LIN {X 0,Y 468.044,Z 554.979,A -85,B 0,C 180,E1 -7471.506,E2 -7471.506} C_VEL
LIN {X 0,Y 468.414,Z 546.131,A -85,B 0,C 180,E1 -7472.58,E2 -7472.58} C_VEL
LIN {X 0,Y 468.833,Z 536.407,A -85,B 0,C 180,E1 -7473.545,E2 -7473.545} C_VEL
LIN {X 0,Y 469.337,Z 525.651,A -85,B 0,C 180,E1 -7474.401,E2 -7474.401} C_VEL
LIN {X 0,Y 469.768,Z 513.644,A -85,B 0,C 180,E1 -7475.15,E2 -7475.15} C_VEL
LIN {X 0,Y 470.118,Z 501.093,A -85,B 0,C 180,E1 -7475.738,E2 -7475.738} C_VEL
LIN {X 0,Y 470.387,Z 488.653,A -85,B 0,C 180,E1 -7476.138,E2 -7476.138} C_VEL
LIN {X 0,Y 470.656,Z 471.073,A -85,B 0,C 180,E1 -7476.457,E2 -7476.457} C_VEL
LIN {X 0,Y 471.201,Z 391.14,A -85,B 0,C 180,E1 -7477.679,E2 -7477.679} C_VEL
LIN {X 0,Y 468.508,Z 378.211,A -85,B 0,C 180,E1 -7477.998,E2 -7477.998} C_VEL
LIN {X 0,Y 468.62,Z 369.536,A -85,B 0,C 180,E1 -7479.931,E2 -7479.931} C_VEL
LIN {X 0,Y 467.725,Z 363.226,A -85,B 0,C 180,E1 -7481.429,E2 -7481.429} C_VEL
LIN {X 0,Y 467.612,Z 363.236,A -85,B 0,C 180,E1 -7484.803,E2 -7484.803} C_VEL
LIN {X 0,Y 467.612,Z 363.233,A -85,B 0,C 180,E1 -7487.493,E2 -7487.493} C_VEL
LIN {X 0,Y 467.627,Z 363.237,A -85,B 0,C 180,E1 -7490.222,E2 -7490.222} C_VEL
LIN {X 0,Y 467.577,Z 363.241,A -85,B 0,C 180,E1 -7493.942,E2 -7493.942} C_VEL
LIN {X 0,Y 467.62,Z 363.234,A -85,B 0,C 180,E1 -7496.799,E2 -7496.799} C_VEL
LIN {X 0,Y 467.59,Z 363.239,A -85,B 0,C 180,E1 -7499.735,E2 -7499.735} C_VEL
LIN {X 0,Y 467.585,Z 363.239,A -85,B 0,C 180,E1 -7502.757,E2 -7502.757} C_VEL
LIN {X 0,Y 467.557,Z 363.244,A -85,B 0,C 180,E1 -7505.888,E2 -7505.888} C_VEL
LIN {X 0,Y 467.582,Z 363.239,A -85,B 0,C 180,E1 -7509.144,E2 -7509.144} C_VEL
LIN {X 0,Y 467.585,Z 363.239,A -85,B 0,C 180,E1 -7512.566,E2 -7512.566} C_VEL
LIN {X 0,Y 467.568,Z 363.241,A -85,B 0,C 180,E1 -7515.052,E2 -7515.052} C_VEL
LIN {X 0,Y 467.622,Z 363.235,A -85,B 0,C 180,E1 -7517.443,E2 -7517.443} C_VEL
LIN {X 0,Y 467.611,Z 363.236,A -85,B 0,C 180,E1 -7520.858,E2 -7520.858} C_VEL
LIN {X 0,Y 467.558,Z 363.244,A -85,B 0,C 180,E1 -7524.26,E2 -7524.26} C_VEL
LIN {X 0,Y 467.577,Z 363.241,A -85,B 0,C 180,E1 -7527.32,E2 -7527.32} C_VEL
LIN {X 0,Y 467.564,Z 363.242,A -85,B 0,C 180,E1 -7530.666,E2 -7530.666} C_VEL
LIN {X 0,Y 467.622,Z 363.236,A -85,B 0,C 180,E1 -7533.2,E2 -7533.2} C_VEL
LIN {X 0,Y 467.587,Z 363.239,A -85,B 0,C 180,E1 -7536.467,E2 -7536.467} C_VEL
LIN {X 0,Y 467.618,Z 363.238,A -85,B 0,C 180,E1 -7539.777,E2 -7539.777} C_VEL
LIN {X 0,Y 467.602,Z 363.238,A -85,B 0,C 180,E1 -7542.506,E2 -7542.506} C_VEL
LIN {X 0,Y 467.602,Z 363.239,A -85,B 0,C 180,E1 -7545.196,E2 -7545.196} C_VEL
LIN {X 0,Y 467.689,Z 363.228,A -85,B 0,C 180,E1 -7547.855,E2 -7547.855} C_VEL
LIN {X 0,Y 467.674,Z 363.23,A -85,B 0,C 180,E1 -7551.357,E2 -7551.357} C_VEL
LIN {X 0,Y 467.735,Z 363.221,A -85,B 0,C 180,E1 -7553.962,E2 -7553.962} C_VEL
LIN {X 0,Y 467.853,Z 363.208,A -85,B 0,C 180,E1 -7557.417,E2 -7557.417} C_VEL
LIN {X 0,Y 467.873,Z 363.203,A -85,B 0,C 180,E1 -7560,E2 -7560} C_VEL
LIN {X 0,Y 467.853,Z 363.209,A -85,B 0,C 180,E1 -7562.583,E2 -7562.583} C_VEL
LIN {X 0,Y 467.739,Z 363.22,A -85,B 0,C 180,E1 -7566.037,E2 -7566.037} C_VEL
LIN {X 0,Y 467.674,Z 363.231,A -85,B 0,C 180,E1 -7568.643,E2 -7568.643} C_VEL
LIN {X 0,Y 467.682,Z 363.23,A -85,B 0,C 180,E1 -7572.379,E2 -7572.379} C_VEL
LIN {X 0,Y 467.64,Z 363.232,A -85,B 0,C 180,E1 -7575.886,E2 -7575.886} C_VEL
LIN {X 0,Y 467.615,Z 363.236,A -85,B 0,C 180,E1 -7579.308,E2 -7579.308} C_VEL
LIN {X 0,Y 467.541,Z 363.246,A -85,B 0,C 180,E1 -7582.073,E2 -7582.073} C_VEL
LIN {X 0,Y 467.597,Z 363.238,A -85,B 0,C 180,E1 -7584.888,E2 -7584.888} C_VEL
LIN {X 0,Y 467.62,Z 363.235,A -85,B 0,C 180,E1 -7587.769,E2 -7587.769} C_VEL
LIN {X 0,Y 467.562,Z 363.242,A -85,B 0,C 180,E1 -7591.046,E2 -7591.046} C_VEL
LIN {X 0,Y 467.584,Z 363.244,A -85,B 0,C 180,E1 -7594.243,E2 -7594.243} C_VEL
LIN {X 0,Y 467.545,Z 363.243,A -85,B 0,C 180,E1 -7597.188,E2 -7597.188} C_VEL
LIN {X 0,Y 467.591,Z 363.242,A -85,B 0,C 180,E1 -7600.263,E2 -7600.263} C_VEL
LIN {X 0,Y 467.614,Z 363.236,A -85,B 0,C 180,E1 -7602.572,E2 -7602.572} C_VEL
LIN {X 0,Y 467.566,Z 363.24,A -85,B 0,C 180,E1 -7605.054,E2 -7605.054} C_VEL
LIN {X 0,Y 467.585,Z 363.238,A -85,B 0,C 180,E1 -7607.441,E2 -7607.441} C_VEL
LIN {X 0,Y 467.579,Z 363.238,A -85,B 0,C 180,E1 -7610.856,E2 -7610.856} C_VEL
LIN {X 0,Y 467.561,Z 363.243,A -85,B 0,C 180,E1 -7614.261,E2 -7614.261} C_VEL
LIN {X 0,Y 467.581,Z 363.238,A -85,B 0,C 180,E1 -7617.321,E2 -7617.321} C_VEL
LIN {X 0,Y 467.578,Z 363.24,A -85,B 0,C 180,E1 -7620.666,E2 -7620.666} C_VEL
LIN {X 0,Y 467.657,Z 363.297,A -85,B 0,C 180,E1 -7623.474,E2 -7623.474} C_VEL
LIN {X 0,Y 470.033,Z 375.942,A -85,B 0,C 180,E1 -7625.795,E2 -7625.795} C_VEL
LIN {X 0,Y 469.281,Z 393.239,A -85,B 0,C 180,E1 -7628.731,E2 -7628.731} C_VEL
LIN {X 0,Y 468.542,Z 411.912,A -85,B 0,C 180,E1 -7631.866,E2 -7631.866} C_VEL
LIN {X 0,Y 468.286,Z 419.154,A -85,B 0,C 180,E1 -7633.033,E2 -7633.033} C_VEL
LIN {X 0,Y 471.101,Z 439.527,A -85,B 0,C 180,E1 -7633.442,E2 -7633.442} C_VEL
LIN {X 0,Y 470.448,Z 528.104,A -85,B 0,C 180,E1 -7634.818,E2 -7634.818} C_VEL
LIN {X 0,Y 470.07,Z 541.203,A -85,B 0,C 180,E1 -7635.193,E2 -7635.193} C_VEL
LIN {X 0,Y 469.613,Z 553.288,A -85,B 0,C 180,E1 -7635.704,E2 -7635.704} C_VEL
LIN {X 0,Y 469.161,Z 564.699,A -85,B 0,C 180,E1 -7636.354,E2 -7636.354} C_VEL
LIN {X 0,Y 468.609,Z 576.212,A -85,B 0,C 180,E1 -7637.2,E2 -7637.2} C_VEL
LIN {X 0,Y 468.197,Z 587.011,A -85,B 0,C 180,E1 -7638.199,E2 -7638.199} C_VEL
LIN {X 0,Y 467.767,Z 595.641,A -85,B 0,C 180,E1 -7639.175,E2 -7639.175} C_VEL
LIN {X 0,Y 467.401,Z 603.6,A -85,B 0,C 180,E1 -7640.261,E2 -7640.261} C_VEL
LIN {X 0,Y 467.103,Z 611.375,A -85,B 0,C 180,E1 -7641.565,E2 -7641.565} C_VEL
LIN {X 0,Y 466.858,Z 618.527,A -85,B 0,C 180,E1 -7643.083,E2 -7643.083} C_VEL
LIN {X 0,Y 466.762,Z 623.289,A -85,B 0,C 180,E1 -7644.384,E2 -7644.384} C_VEL
LIN {X 0,Y 466.658,Z 626.925,A -85,B 0,C 180,E1 -7645.682,E2 -7645.682} C_VEL
LIN {X 0,Y 466.712,Z 628.806,A -85,B 0,C 180,E1 -7646.547,E2 -7646.547} C_VEL
LIN {X 0,Y 466.68,Z 630.213,A -85,B 0,C 180,E1 -7647.411,E2 -7647.411} C_VEL
LIN {X 0,Y 466.661,Z 631.215,A -85,B 0,C 180,E1 -7648.274,E2 -7648.274} C_VEL
LIN {X 0,Y 466.6,Z 632.044,A -85,B 0,C 180,E1 -7650,E2 -7650} C_VEL
LIN {X 0,Y 466.62,Z 631.83,A -85,B 0,C 180,E1 -7650.863,E2 -7650.863} C_VEL
LIN {X 0,Y 466.661,Z 631.221,A -85,B 0,C 180,E1 -7651.726,E2 -7651.726} C_VEL
LIN {X 0,Y 466.68,Z 630.222,A -85,B 0,C 180,E1 -7652.589,E2 -7652.589} C_VEL
LIN {X 0,Y 466.697,Z 628.821,A -85,B 0,C 180,E1 -7653.453,E2 -7653.453} C_VEL
LIN {X 0,Y 466.69,Z 625.873,A -85,B 0,C 180,E1 -7654.751,E2 -7654.751} C_VEL
LIN {X 0,Y 466.751,Z 621.888,A -85,B 0,C 180,E1 -7656.05,E2 -7656.05} C_VEL
LIN {X 0,Y 466.942,Z 615.771,A -85,B 0,C 180,E1 -7657.568,E2 -7657.568} C_VEL
LIN {X 0,Y 467.152,Z 609.091,A -85,B 0,C 180,E1 -7658.87,E2 -7658.87} C_VEL
LIN {X 0,Y 467.496,Z 600.812,A -85,B 0,C 180,E1 -7660.174,E2 -7660.174} C_VEL
LIN {X 0,Y 467.987,Z 592.352,A -85,B 0,C 180,E1 -7661.258,E2 -7661.258} C_VEL
LIN {X 0,Y 468.464,Z 582.434,A -85,B 0,C 180,E1 -7662.295,E2 -7662.295} C_VEL
LIN {X 0,Y 468.902,Z 571.605,A -85,B 0,C 180,E1 -7663.213,E2 -7663.213} C_VEL
LIN {X 0,Y 469.437,Z 560.342,A -85,B 0,C 180,E1 -7663.969,E2 -7663.969} C_VEL
LIN {X 0,Y 469.903,Z 548.916,A -85,B 0,C 180,E1 -7664.563,E2 -7664.563} C_VEL
LIN {X 0,Y 470.368,Z 535.882,A -85,B 0,C 180,E1 -7665.046,E2 -7665.046} C_VEL
LIN {X 0,Y 470.678,Z 521.948,A -85,B 0,C 180,E1 -7665.369,E2 -7665.369} C_VEL
LIN {X 0,Y 471.166,Z 437.424,A -85,B 0,C 180,E1 -7666.676,E2 -7666.676} C_VEL
LIN {X 0,Y 468.328,Z 418.62,A -85,B 0,C 180,E1 -7667.1,E2 -7667.1} C_VEL
LIN {X 0,Y 469.117,Z 400.586,A -85,B 0,C 180,E1 -7670.155,E2 -7670.155} C_VEL
LIN {X 0,Y 470.064,Z 380.743,A -85,B 0,C 180,E1 -7673.574,E2 -7673.574} C_VEL
LIN {X 0,Y 470.181,Z 375.849,A -85,B 0,C 180,E1 -7674.436,E2 -7674.436} C_VEL
LIN {X 0,Y 467.689,Z 363.253,A -85,B 0,C 180,E1 -7676.851,E2 -7676.851} C_VEL
LIN {X 0,Y 467.587,Z 363.239,A -85,B 0,C 180,E1 -7679.735,E2 -7679.735} C_VEL
LIN {X 0,Y 467.582,Z 363.239,A -85,B 0,C 180,E1 -7682.758,E2 -7682.758} C_VEL
LIN {X 0,Y 467.555,Z 363.247,A -85,B 0,C 180,E1 -7685.889,E2 -7685.889} C_VEL
LIN {X 0,Y 467.579,Z 363.238,A -85,B 0,C 180,E1 -7689.144,E2 -7689.144} C_VEL
LIN {X 0,Y 467.582,Z 363.236,A -85,B 0,C 180,E1 -7692.566,E2 -7692.566} C_VEL
LIN {X 0,Y 467.566,Z 363.238,A -85,B 0,C 180,E1 -7695.052,E2 -7695.052} C_VEL
LIN {X 0,Y 467.619,Z 363.235,A -85,B 0,C 180,E1 -7697.443,E2 -7697.443} C_VEL
LIN {X 0,Y 467.594,Z 363.234,A -85,B 0,C 180,E1 -7700.856,E2 -7700.856} C_VEL
LIN {X 0,Y 467.557,Z 363.24,A -85,B 0,C 180,E1 -7704.26,E2 -7704.26} C_VEL
LIN {X 0,Y 467.575,Z 363.243,A -85,B 0,C 180,E1 -7707.32,E2 -7707.32} C_VEL
LIN {X 0,Y 467.571,Z 363.238,A -85,B 0,C 180,E1 -7710.665,E2 -7710.665} C_VEL
LIN {X 0,Y 467.62,Z 363.236,A -85,B 0,C 180,E1 -7713.2,E2 -7713.2} C_VEL
LIN {X 0,Y 467.585,Z 363.231,A -85,B 0,C 180,E1 -7716.467,E2 -7716.467} C_VEL
LIN {X 0,Y 467.616,Z 363.233,A -85,B 0,C 180,E1 -7719.777,E2 -7719.777} C_VEL
LIN {X 0,Y 467.601,Z 363.235,A -85,B 0,C 180,E1 -7722.507,E2 -7722.507} C_VEL
LIN {X 0,Y 467.598,Z 363.238,A -85,B 0,C 180,E1 -7725.196,E2 -7725.196} C_VEL
LIN {X 0,Y 467.673,Z 363.226,A -85,B 0,C 180,E1 -7727.855,E2 -7727.855} C_VEL
LIN {X 0,Y 467.674,Z 363.23,A -85,B 0,C 180,E1 -7731.357,E2 -7731.357} C_VEL
LIN {X 0,Y 467.735,Z 363.214,A -85,B 0,C 180,E1 -7733.963,E2 -7733.963} C_VEL
LIN {X 0,Y 467.853,Z 363.204,A -85,B 0,C 180,E1 -7737.417,E2 -7737.417} C_VEL
LIN {X 0,Y 467.873,Z 363.2,A -85,B 0,C 180,E1 -7740,E2 -7740} C_VEL
LIN {X 0,Y 467.853,Z 363.208,A -85,B 0,C 180,E1 -7742.583,E2 -7742.583} C_VEL
LIN {X 0,Y 467.736,Z 363.219,A -85,B 0,C 180,E1 -7746.038,E2 -7746.038} C_VEL
LIN {X 0,Y 467.674,Z 363.228,A -85,B 0,C 180,E1 -7748.643,E2 -7748.643} C_VEL
LIN {X 0,Y 467.648,Z 363.23,A -85,B 0,C 180,E1 -7752.146,E2 -7752.146} C_VEL
LIN {X 0,Y 467.631,Z 363.231,A -85,B 0,C 180,E1 -7755.696,E2 -7755.696} C_VEL
LIN {X 0,Y 467.61,Z 363.238,A -85,B 0,C 180,E1 -7758.765,E2 -7758.765} C_VEL
LIN {X 0,Y 467.573,Z 363.236,A -85,B 0,C 180,E1 -7761.269,E2 -7761.269} C_VEL
LIN {X 0,Y 467.567,Z 363.242,A -85,B 0,C 180,E1 -7763.944,E2 -7763.944} C_VEL
LIN {X 0,Y 467.621,Z 363.228,A -85,B 0,C 180,E1 -7766.8,E2 -7766.8} C_VEL
LIN {X 0,Y 467.548,Z 363.243,A -85,B 0,C 180,E1 -7769.739,E2 -7769.739} C_VEL
LIN {X 0,Y 467.579,Z 363.239,A -85,B 0,C 180,E1 -7772.759,E2 -7772.759} C_VEL
LIN {X 0,Y 467.552,Z 363.246,A -85,B 0,C 180,E1 -7775.89,E2 -7775.89} C_VEL
LIN {X 0,Y 467.596,Z 363.236,A -85,B 0,C 180,E1 -7779.144,E2 -7779.144} C_VEL
LIN {X 0,Y 467.617,Z 363.234,A -85,B 0,C 180,E1 -7782.572,E2 -7782.572} C_VEL
LIN {X 0,Y 467.568,Z 363.243,A -85,B 0,C 180,E1 -7785.054,E2 -7785.054} C_VEL
LIN {X 0,Y 467.587,Z 363.241,A -85,B 0,C 180,E1 -7787.441,E2 -7787.441} C_VEL
LIN {X 0,Y 467.619,Z 363.235,A -85,B 0,C 180,E1 -7790.86,E2 -7790.86} C_VEL
LIN {X 0,Y 467.564,Z 363.244,A -85,B 0,C 180,E1 -7794.261,E2 -7794.261} C_VEL
LIN {X 0,Y 467.583,Z 363.241,A -85,B 0,C 180,E1 -7797.322,E2 -7797.322} C_VEL
LIN {X 0,Y 467.645,Z 363.312,A -85,B 0,C 180,E1 -7800.441,E2 -7800.441} C_VEL
LIN {X 0,Y 468.864,Z 370.492,A -85,B 0,C 180,E1 -7802.176,E2 -7802.176} C_VEL
LIN {X 0,Y 468.609,Z 378.685,A -85,B 0,C 180,E1 -7803.992,E2 -7803.992} C_VEL
LIN {X 0,Y 471.605,Z 392.631,A -85,B 0,C 180,E1 -7804.336,E2 -7804.336} C_VEL
LIN {X 0,Y 470.941,Z 465.261,A -85,B 0,C 180,E1 -7805.452,E2 -7805.452} C_VEL
LIN {X 0,Y 470.243,Z 471.119,A -85,B 0,C 180,E1 -7805.515,E2 -7805.515} C_VEL
LIN {X 0,Y 464.863,Z 488.149,A -85,B 0,C 180,E1 -7805.631,E2 -7805.631} C_VEL
LIN {X 0,Y 463.849,Z 493.862,A -85,B 0,C 180,E1 -7805.755,E2 -7805.755} C_VEL
LIN {X 0,Y 463.78,Z 495.764,A -85,B 0,C 180,E1 -7805.814,E2 -7805.814} C_VEL
LIN {X 0,Y 463.399,Z 507.867,A -85,B 0,C 180,E1 -7806.303,E2 -7806.303} C_VEL
LIN {X 0,Y 462.962,Z 520.228,A -85,B 0,C 180,E1 -7806.99,E2 -7806.99} C_VEL
LIN {X 0,Y 462.512,Z 531.401,A -85,B 0,C 180,E1 -7807.796,E2 -7807.796} C_VEL
LIN {X 0,Y 461.866,Z 542.532,A -85,B 0,C 180,E1 -7808.815,E2 -7808.815} C_VEL
LIN {X 0,Y 461.322,Z 552.494,A -85,B 0,C 180,E1 -7809.954,E2 -7809.954} C_VEL
LIN {X 0,Y 460.873,Z 560.782,A -85,B 0,C 180,E1 -7811.121,E2 -7811.121} C_VEL
LIN {X 0,Y 460.441,Z 568.432,A -85,B 0,C 180,E1 -7812.455,E2 -7812.455} C_VEL
LIN {X 0,Y 460.171,Z 573.745,A -85,B 0,C 180,E1 -7813.588,E2 -7813.588} C_VEL
LIN {X 0,Y 459.945,Z 578.843,A -85,B 0,C 180,E1 -7814.944,E2 -7814.944} C_VEL
LIN {X 0,Y 459.752,Z 582.757,A -85,B 0,C 180,E1 -7816.294,E2 -7816.294} C_VEL
LIN {X 0,Y 459.658,Z 586.366,A -85,B 0,C 180,E1 -7818.11,E2 -7818.11} C_VEL
LIN {X 0,Y 459.576,Z 587.863,A -85,B 0,C 180,E1 -7819.426,E2 -7819.426} C_VEL
LIN {X 0,Y 459.494,Z 588.394,A -85,B 0,C 180,E1 -7820.314,E2 -7820.314} C_VEL
LIN {X 0,Y 459.53,Z 588.483,A -85,B 0,C 180,E1 -7821.203,E2 -7821.203} C_VEL
LIN {X 0,Y 459.618,Z 587.497,A -85,B 0,C 180,E1 -7822.974,E2 -7822.974} C_VEL
LIN {X 0,Y 459.67,Z 586.415,A -85,B 0,C 180,E1 -7823.856,E2 -7823.856} C_VEL
LIN {X 0,Y 459.672,Z 584.89,A -85,B 0,C 180,E1 -7824.737,E2 -7824.737} C_VEL
LIN {X 0,Y 459.809,Z 581.826,A -85,B 0,C 180,E1 -7826.056,E2 -7826.056} C_VEL
LIN {X 0,Y 459.921,Z 577.728,A -85,B 0,C 180,E1 -7827.373,E2 -7827.373} C_VEL
LIN {X 0,Y 460.167,Z 571.478,A -85,B 0,C 180,E1 -7828.906,E2 -7828.906} C_VEL
LIN {X 0,Y 460.547,Z 564.676,A -85,B 0,C 180,E1 -7830.219,E2 -7830.219} C_VEL
LIN {X 0,Y 460.992,Z 556.186,A -85,B 0,C 180,E1 -7831.529,E2 -7831.529} C_VEL
LIN {X 0,Y 461.388,Z 547.502,A -85,B 0,C 180,E1 -7832.619,E2 -7832.619} C_VEL
LIN {X 0,Y 461.814,Z 537.987,A -85,B 0,C 180,E1 -7833.599,E2 -7833.599} C_VEL
LIN {X 0,Y 462.373,Z 527.564,A -85,B 0,C 180,E1 -7834.468,E2 -7834.468} C_VEL
LIN {X 0,Y 462.838,Z 516.054,A -85,B 0,C 180,E1 -7835.227,E2 -7835.227} C_VEL
LIN {X 0,Y 463.103,Z 504.183,A -85,B 0,C 180,E1 -7835.825,E2 -7835.825} C_VEL
LIN {X 0,Y 463.473,Z 491.224,A -85,B 0,C 180,E1 -7836.284,E2 -7836.284} C_VEL
LIN {X 0,Y 463.727,Z 478.883,A -85,B 0,C 180,E1 -7836.554,E2 -7836.554} C_VEL
LIN {X 0,Y 464.385,Z 392.218,A -85,B 0,C 180,E1 -7837.897,E2 -7837.897} C_VEL
LIN {X 0,Y 461.564,Z 378.518,A -85,B 0,C 180,E1 -7838.237,E2 -7838.237} C_VEL
LIN {X 0,Y 461.621,Z 370.343,A -85,B 0,C 180,E1 -7840.083,E2 -7840.083} C_VEL
LIN {X 0,Y 460.663,Z 364.106,A -85,B 0,C 180,E1 -7841.606,E2 -7841.606} C_VEL
LIN {X 0,Y 460.575,Z 364.111,A -85,B 0,C 180,E1 -7845.034,E2 -7845.034} C_VEL
LIN {X 0,Y 460.562,Z 364.113,A -85,B 0,C 180,E1 -7847.769,E2 -7847.769} C_VEL
LIN {X 0,Y 460.556,Z 364.117,A -85,B 0,C 180,E1 -7850.547,E2 -7850.547} C_VEL
LIN {X 0,Y 460.541,Z 364.116,A -85,B 0,C 180,E1 -7853.705,E2 -7853.705} C_VEL
LIN {X 0,Y 460.566,Z 364.118,A -85,B 0,C 180,E1 -7856.264,E2 -7856.264} C_VEL
LIN {X 0,Y 460.55,Z 364.114,A -85,B 0,C 180,E1 -7859.229,E2 -7859.229} C_VEL
LIN {X 0,Y 460.534,Z 364.122,A -85,B 0,C 180,E1 -7862.283,E2 -7862.283} C_VEL
LIN {X 0,Y 460.514,Z 364.119,A -85,B 0,C 180,E1 -7865.444,E2 -7865.444} C_VEL
LIN {X 0,Y 460.545,Z 364.115,A -85,B 0,C 180,E1 -7868.897,E2 -7868.897} C_VEL
LIN {X 0,Y 460.521,Z 364.123,A -85,B 0,C 180,E1 -7872.18,E2 -7872.18} C_VEL
LIN {X 0,Y 460.52,Z 364.119,A -85,B 0,C 180,E1 -7875.411,E2 -7875.411} C_VEL
LIN {X 0,Y 460.542,Z 364.117,A -85,B 0,C 180,E1 -7878.395,E2 -7878.395} C_VEL
LIN {X 0,Y 460.54,Z 364.117,A -85,B 0,C 180,E1 -7881.268,E2 -7881.268} C_VEL
LIN {X 0,Y 460.508,Z 364.121,A -85,B 0,C 180,E1 -7884.554,E2 -7884.554} C_VEL
LIN {X 0,Y 460.527,Z 364.121,A -85,B 0,C 180,E1 -7887.715,E2 -7887.715} C_VEL
LIN {X 0,Y 460.534,Z 364.118,A -85,B 0,C 180,E1 -7890.768,E2 -7890.768} C_VEL
LIN {X 0,Y 460.562,Z 364.117,A -85,B 0,C 180,E1 -7893.734,E2 -7893.734} C_VEL
LIN {X 0,Y 460.541,Z 364.117,A -85,B 0,C 180,E1 -7896.623,E2 -7896.623} C_VEL
LIN {X 0,Y 460.564,Z 364.115,A -85,B 0,C 180,E1 -7899.453,E2 -7899.453} C_VEL
LIN {X 0,Y 460.552,Z 364.116,A -85,B 0,C 180,E1 -7902.23,E2 -7902.23} C_VEL
LIN {X 0,Y 460.56,Z 364.116,A -85,B 0,C 180,E1 -7904.964,E2 -7904.964} C_VEL
LIN {X 0,Y 460.649,Z 364.106,A -85,B 0,C 180,E1 -7907.667,E2 -7907.667} C_VEL
LIN {X 0,Y 460.621,Z 364.108,A -85,B 0,C 180,E1 -7911.223,E2 -7911.223} C_VEL
LIN {X 0,Y 460.701,Z 364.098,A -85,B 0,C 180,E1 -7913.87,E2 -7913.87} C_VEL
LIN {X 0,Y 460.818,Z 364.084,A -85,B 0,C 180,E1 -7917.377,E2 -7917.377} C_VEL
LIN {X 0,Y 460.844,Z 364.079,A -85,B 0,C 180,E1 -7920,E2 -7920} C_VEL
LIN {X 0,Y 460.818,Z 364.085,A -85,B 0,C 180,E1 -7922.622,E2 -7922.622} C_VEL
LIN {X 0,Y 460.704,Z 364.097,A -85,B 0,C 180,E1 -7926.13,E2 -7926.13} C_VEL
LIN {X 0,Y 460.621,Z 364.109,A -85,B 0,C 180,E1 -7928.776,E2 -7928.776} C_VEL
LIN {X 0,Y 460.625,Z 364.11,A -85,B 0,C 180,E1 -7932.457,E2 -7932.457} C_VEL
LIN {X 0,Y 460.591,Z 364.111,A -85,B 0,C 180,E1 -7935.998,E2 -7935.998} C_VEL
LIN {X 0,Y 460.562,Z 364.115,A -85,B 0,C 180,E1 -7938.902,E2 -7938.902} C_VEL
LIN {X 0,Y 460.553,Z 364.115,A -85,B 0,C 180,E1 -7941.484,E2 -7941.484} C_VEL
LIN {X 0,Y 460.536,Z 364.121,A -85,B 0,C 180,E1 -7944.333,E2 -7944.333} C_VEL
LIN {X 0,Y 460.576,Z 364.113,A -85,B 0,C 180,E1 -7947.244,E2 -7947.244} C_VEL
LIN {X 0,Y 460.503,Z 364.126,A -85,B 0,C 180,E1 -7950.24,E2 -7950.24} C_VEL
LIN {X 0,Y 460.523,Z 364.118,A -85,B 0,C 180,E1 -7953.325,E2 -7953.325} C_VEL
LIN {X 0,Y 460.473,Z 364.126,A -85,B 0,C 180,E1 -7956.53,E2 -7956.53} C_VEL
LIN {X 0,Y 460.57,Z 364.115,A -85,B 0,C 180,E1 -7959.858,E2 -7959.858} C_VEL
LIN {X 0,Y 460.537,Z 364.116,A -85,B 0,C 180,E1 -7962.905,E2 -7962.905} C_VEL
LIN {X 0,Y 460.507,Z 364.123,A -85,B 0,C 180,E1 -7965.831,E2 -7965.831} C_VEL
LIN {X 0,Y 460.527,Z 364.117,A -85,B 0,C 180,E1 -7968.99,E2 -7968.99} C_VEL
LIN {X 0,Y 460.524,Z 364.117,A -85,B 0,C 180,E1 -7971.268,E2 -7971.268} C_VEL
LIN {X 0,Y 460.512,Z 364.119,A -85,B 0,C 180,E1 -7974.555,E2 -7974.555} C_VEL
LIN {X 0,Y 460.532,Z 364.12,A -85,B 0,C 180,E1 -7977.716,E2 -7977.716} C_VEL
LIN {X 0,Y 460.547,Z 364.116,A -85,B 0,C 180,E1 -7980.77,E2 -7980.77} C_VEL
LIN {X 0,Y 460.606,Z 364.146,A -85,B 0,C 180,E1 -7983.28,E2 -7983.28} C_VEL
LIN {X 0,Y 463.027,Z 376.596,A -85,B 0,C 180,E1 -7985.603,E2 -7985.603} C_VEL
LIN {X 0,Y 462.428,Z 392.07,A -85,B 0,C 180,E1 -7988.277,E2 -7988.277} C_VEL
LIN {X 0,Y 461.503,Z 412.791,A -85,B 0,C 180,E1 -7991.81,E2 -7991.81} C_VEL
LIN {X 0,Y 461.27,Z 418.674,A -85,B 0,C 180,E1 -7992.787,E2 -7992.787} C_VEL
LIN {X 0,Y 464.252,Z 439.85,A -85,B 0,C 180,E1 -7993.222,E2 -7993.222} C_VEL
LIN {X 0,Y 463.581,Z 526.961,A -85,B 0,C 180,E1 -7994.587,E2 -7994.587} C_VEL
LIN {X 0,Y 463.208,Z 540.34,A -85,B 0,C 180,E1 -7994.969,E2 -7994.969} C_VEL
LIN {X 0,Y 462.727,Z 552.571,A -85,B 0,C 180,E1 -7995.487,E2 -7995.487} C_VEL
LIN {X 0,Y 462.217,Z 564.087,A -85,B 0,C 180,E1 -7996.145,E2 -7996.145} C_VEL
LIN {X 0,Y 461.665,Z 575.364,A -85,B 0,C 180,E1 -7996.978,E2 -7996.978} C_VEL
LIN {X 0,Y 461.16,Z 586.507,A -85,B 0,C 180,E1 -7998.016,E2 -7998.016} C_VEL
LIN {X 0,Y 460.764,Z 595.173,A -85,B 0,C 180,E1 -7999.009,E2 -7999.009} C_VEL
LIN {X 0,Y 460.349,Z 603.157,A -85,B 0,C 180,E1 -8000.111,E2 -8000.111} C_VEL
LIN {X 0,Y 460.031,Z 610.965,A -85,B 0,C 180,E1 -8001.434,E2 -8001.434} C_VEL
LIN {X 0,Y 459.774,Z 618.134,A -85,B 0,C 180,E1 -8002.976,E2 -8002.976} C_VEL
LIN {X 0,Y 459.659,Z 622.91,A -85,B 0,C 180,E1 -8004.297,E2 -8004.297} C_VEL
LIN {X 0,Y 459.573,Z 626.56,A -85,B 0,C 180,E1 -8005.615,E2 -8005.615} C_VEL
LIN {X 0,Y 459.609,Z 628.448,A -85,B 0,C 180,E1 -8006.493,E2 -8006.493} C_VEL
LIN {X 0,Y 459.602,Z 629.864,A -85,B 0,C 180,E1 -8007.371,E2 -8007.371} C_VEL
LIN {X 0,Y 459.553,Z 631.486,A -85,B 0,C 180,E1 -8009.124,E2 -8009.124} C_VEL
LIN {X 0,Y 459.532,Z 631.711,A -85,B 0,C 180,E1 -8010,E2 -8010} C_VEL
LIN {X 0,Y 459.553,Z 631.504,A -85,B 0,C 180,E1 -8010.876,E2 -8010.876} C_VEL
LIN {X 0,Y 459.601,Z 629.904,A -85,B 0,C 180,E1 -8012.629,E2 -8012.629} C_VEL
LIN {X 0,Y 459.594,Z 628.508,A -85,B 0,C 180,E1 -8013.507,E2 -8013.507} C_VEL
LIN {X 0,Y 459.621,Z 625.57,A -85,B 0,C 180,E1 -8014.824,E2 -8014.824} C_VEL
LIN {X 0,Y 459.714,Z 620.574,A -85,B 0,C 180,E1 -8016.431,E2 -8016.431} C_VEL
LIN {X 0,Y 459.89,Z 614.487,A -85,B 0,C 180,E1 -8017.905,E2 -8017.905} C_VEL
LIN {X 0,Y 460.171,Z 607.602,A -85,B 0,C 180,E1 -8019.228,E2 -8019.228} C_VEL
LIN {X 0,Y 460.571,Z 599.022,A -85,B 0,C 180,E1 -8020.551,E2 -8020.551} C_VEL
LIN {X 0,Y 461.072,Z 590.225,A -85,B 0,C 180,E1 -8021.652,E2 -8021.652} C_VEL
LIN {X 0,Y 461.547,Z 579.698,A -85,B 0,C 180,E1 -8022.728,E2 -8022.728} C_VEL
LIN {X 0,Y 462.145,Z 568.617,A -85,B 0,C 180,E1 -8023.633,E2 -8023.633} C_VEL
LIN {X 0,Y 462.688,Z 556.514,A -85,B 0,C 180,E1 -8024.402,E2 -8024.402} C_VEL
LIN {X 0,Y 463.272,Z 543.889,A -85,B 0,C 180,E1 -8025.001,E2 -8025.001} C_VEL
LIN {X 0,Y 463.697,Z 531.564,A -85,B 0,C 180,E1 -8025.409,E2 -8025.409} C_VEL
LIN {X 0,Y 463.92,Z 515.932,A -85,B 0,C 180,E1 -8025.711,E2 -8025.711} C_VEL
LIN {X 0,Y 464.424,Z 438.295,A -85,B 0,C 180,E1 -8026.929,E2 -8026.929} C_VEL
LIN {X 0,Y 461.386,Z 418.289,A -85,B 0,C 180,E1 -8027.389,E2 -8027.389} C_VEL
LIN {X 0,Y 462.193,Z 400.426,A -85,B 0,C 180,E1 -8030.47,E2 -8030.47} C_VEL
LIN {X 0,Y 463.166,Z 381.944,A -85,B 0,C 180,E1 -8033.709,E2 -8033.709} C_VEL
LIN {X 0,Y 463.319,Z 377.648,A -85,B 0,C 180,E1 -8034.477,E2 -8034.477} C_VEL
LIN {X 0,Y 461.039,Z 366.113,A -85,B 0,C 180,E1 -8036.723,E2 -8036.723} C_VEL
LIN {X 0,Y 460.652,Z 364.106,A -85,B 0,C 180,E1 -8037.146,E2 -8037.146} C_VEL
LIN {X 0,Y 460.527,Z 364.12,A -85,B 0,C 180,E1 -8040.238,E2 -8040.238} C_VEL
LIN {X 0,Y 460.528,Z 364.118,A -85,B 0,C 180,E1 -8043.324,E2 -8043.324} C_VEL
LIN {X 0,Y 460.477,Z 364.125,A -85,B 0,C 180,E1 -8046.528,E2 -8046.528} C_VEL
LIN {X 0,Y 460.555,Z 364.118,A -85,B 0,C 180,E1 -8049.859,E2 -8049.859} C_VEL
LIN {X 0,Y 460.509,Z 364.117,A -85,B 0,C 180,E1 -8052.9,E2 -8052.9} C_VEL
LIN {X 0,Y 460.519,Z 364.121,A -85,B 0,C 180,E1 -8055.828,E2 -8055.828} C_VEL
LIN {X 0,Y 460.538,Z 364.113,A -85,B 0,C 180,E1 -8058.989,E2 -8058.989} C_VEL
LIN {X 0,Y 460.534,Z 364.116,A -85,B 0,C 180,E1 -8061.268,E2 -8061.268} C_VEL
LIN {X 0,Y 460.507,Z 364.117,A -85,B 0,C 180,E1 -8064.554,E2 -8064.554} C_VEL
LIN {X 0,Y 460.526,Z 364.122,A -85,B 0,C 180,E1 -8067.715,E2 -8067.715} C_VEL
LIN {X 0,Y 460.54,Z 364.114,A -85,B 0,C 180,E1 -8070.769,E2 -8070.769} C_VEL
LIN {X 0,Y 460.561,Z 364.106,A -85,B 0,C 180,E1 -8073.735,E2 -8073.735} C_VEL
LIN {X 0,Y 460.539,Z 364.109,A -85,B 0,C 180,E1 -8076.624,E2 -8076.624} C_VEL
LIN {X 0,Y 460.546,Z 364.117,A -85,B 0,C 180,E1 -8079.453,E2 -8079.453} C_VEL
LIN {X 0,Y 460.551,Z 364.113,A -85,B 0,C 180,E1 -8082.23,E2 -8082.23} C_VEL
LIN {X 0,Y 460.557,Z 364.115,A -85,B 0,C 180,E1 -8084.965,E2 -8084.965} C_VEL
LIN {X 0,Y 460.62,Z 364.105,A -85,B 0,C 180,E1 -8087.666,E2 -8087.666} C_VEL
LIN {X 0,Y 460.621,Z 364.11,A -85,B 0,C 180,E1 -8091.224,E2 -8091.224} C_VEL
LIN {X 0,Y 460.701,Z 364.09,A -85,B 0,C 180,E1 -8093.87,E2 -8093.87} C_VEL
LIN {X 0,Y 460.818,Z 364.08,A -85,B 0,C 180,E1 -8097.378,E2 -8097.378} C_VEL
LIN {X 0,Y 460.844,Z 364.075,A -85,B 0,C 180,E1 -8100,E2 -8100} C_VEL
LIN {X 0,Y 460.818,Z 364.085,A -85,B 0,C 180,E1 -8102.623,E2 -8102.623} C_VEL
LIN {X 0,Y 460.702,Z 364.096,A -85,B 0,C 180,E1 -8106.13,E2 -8106.13} C_VEL
LIN {X 0,Y 460.621,Z 364.108,A -85,B 0,C 180,E1 -8108.777,E2 -8108.777} C_VEL
LIN {X 0,Y 460.605,Z 364.109,A -85,B 0,C 180,E1 -8112.445,E2 -8112.445} C_VEL
LIN {X 0,Y 460.592,Z 364.109,A -85,B 0,C 180,E1 -8115.998,E2 -8115.998} C_VEL
LIN {X 0,Y 460.563,Z 364.114,A -85,B 0,C 180,E1 -8118.903,E2 -8118.903} C_VEL
LIN {X 0,Y 460.509,Z 364.116,A -85,B 0,C 180,E1 -8121.486,E2 -8121.486} C_VEL
LIN {X 0,Y 460.536,Z 364.118,A -85,B 0,C 180,E1 -8124.333,E2 -8124.333} C_VEL
LIN {X 0,Y 460.577,Z 364.103,A -85,B 0,C 180,E1 -8127.244,E2 -8127.244} C_VEL
LIN {X 0,Y 460.505,Z 364.125,A -85,B 0,C 180,E1 -8130.241,E2 -8130.241} C_VEL
LIN {X 0,Y 460.525,Z 364.117,A -85,B 0,C 180,E1 -8133.326,E2 -8133.326} C_VEL
LIN {X 0,Y 460.475,Z 364.126,A -85,B 0,C 180,E1 -8136.53,E2 -8136.53} C_VEL
LIN {X 0,Y 460.571,Z 364.116,A -85,B 0,C 180,E1 -8139.859,E2 -8139.859} C_VEL
LIN {X 0,Y 460.54,Z 364.115,A -85,B 0,C 180,E1 -8142.905,E2 -8142.905} C_VEL
LIN {X 0,Y 460.509,Z 364.124,A -85,B 0,C 180,E1 -8145.831,E2 -8145.831} C_VEL
LIN {X 0,Y 460.538,Z 364.118,A -85,B 0,C 180,E1 -8148.991,E2 -8148.991} C_VEL
LIN {X 0,Y 460.547,Z 364.118,A -85,B 0,C 180,E1 -8151.27,E2 -8151.27} C_VEL
LIN {X 0,Y 460.515,Z 364.12,A -85,B 0,C 180,E1 -8154.556,E2 -8154.556} C_VEL
LIN {X 0,Y 460.533,Z 364.122,A -85,B 0,C 180,E1 -8157.717,E2 -8157.717} C_VEL
LIN {X 0,Y 460.607,Z 364.241,A -85,B 0,C 180,E1 -8160.231,E2 -8160.231} C_VEL
LIN {X 0,Y 461.84,Z 371.277,A -85,B 0,C 180,E1 -8161.96,E2 -8161.96} C_VEL
LIN {X 0,Y 461.681,Z 378.848,A -85,B 0,C 180,E1 -8163.699,E2 -8163.699} C_VEL
LIN {X 0,Y 464.892,Z 393.973,A -85,B 0,C 180,E1 -8164.08,E2 -8164.08} C_VEL
LIN {X 0,Y 463.956,Z 485.671,A -85,B 0,C 180,E1 -8165.534,E2 -8165.534} C_VEL
LIN {X 0,Y 463.78,Z 495.764,A -85,B 0,C 180,E1 -8165.814,E2 -8165.814} C_VEL
LIN {X 0,Y 463.118,Z 501.433,A -85,B 0,C 180,E1 -8165.999,E2 -8165.999} C_VEL
LIN {X 0,Y 460.095,Z 510.546,A -85,B 0,C 180,E1 -8166.304,E2 -8166.304} C_VEL
LIN {X 0,Y 456.903,Z 519.371,A -85,B 0,C 180,E1 -8166.7,E2 -8166.7} C_VEL
LIN {X 0,Y 455.983,Z 524.587,A -85,B 0,C 180,E1 -8167.024,E2 -8167.024} C_VEL
LIN {X 0,Y 455.38,Z 535.978,A -85,B 0,C 180,E1 -8167.934,E2 -8167.934} C_VEL
LIN {X 0,Y 454.781,Z 546.065,A -85,B 0,C 180,E1 -8168.944,E2 -8168.944} C_VEL
LIN {X 0,Y 454.232,Z 555.372,A -85,B 0,C 180,E1 -8170.1,E2 -8170.1} C_VEL
LIN {X 0,Y 453.718,Z 564.383,A -85,B 0,C 180,E1 -8171.486,E2 -8171.486} C_VEL
LIN {X 0,Y 453.301,Z 571.518,A -85,B 0,C 180,E1 -8172.868,E2 -8172.868} C_VEL
LIN {X 0,Y 452.956,Z 577.765,A -85,B 0,C 180,E1 -8174.414,E2 -8174.414} C_VEL
LIN {X 0,Y 452.712,Z 582.803,A -85,B 0,C 180,E1 -8176.077,E2 -8176.077} C_VEL
LIN {X 0,Y 452.62,Z 585.737,A -85,B 0,C 180,E1 -8177.445,E2 -8177.445} C_VEL
LIN {X 0,Y 452.573,Z 587.115,A -85,B 0,C 180,E1 -8178.354,E2 -8178.354} C_VEL
LIN {X 0,Y 452.506,Z 588.089,A -85,B 0,C 180,E1 -8179.259,E2 -8179.259} C_VEL
LIN {X 0,Y 452.412,Z 588.673,A -85,B 0,C 180,E1 -8180.161,E2 -8180.161} C_VEL
LIN {X 0,Y 452.439,Z 588.839,A -85,B 0,C 180,E1 -8181.064,E2 -8181.064} C_VEL
LIN {X 0,Y 452.535,Z 587.938,A -85,B 0,C 180,E1 -8182.863,E2 -8182.863} C_VEL
LIN {X 0,Y 452.587,Z 586.911,A -85,B 0,C 180,E1 -8183.76,E2 -8183.76} C_VEL
LIN {X 0,Y 452.603,Z 585.461,A -85,B 0,C 180,E1 -8184.654,E2 -8184.654} C_VEL
LIN {X 0,Y 452.726,Z 582.489,A -85,B 0,C 180,E1 -8185.994,E2 -8185.994} C_VEL
LIN {X 0,Y 452.859,Z 578.486,A -85,B 0,C 180,E1 -8187.332,E2 -8187.332} C_VEL
LIN {X 0,Y 453.021,Z 573.343,A -85,B 0,C 180,E1 -8188.667,E2 -8188.667} C_VEL
LIN {X 0,Y 453.454,Z 566.868,A -85,B 0,C 180,E1 -8190,E2 -8190} C_VEL
LIN {X 0,Y 453.862,Z 558.854,A -85,B 0,C 180,E1 -8191.331,E2 -8191.331} C_VEL
LIN {X 0,Y 454.271,Z 550.681,A -85,B 0,C 180,E1 -8192.438,E2 -8192.438} C_VEL
LIN {X 0,Y 454.728,Z 540.697,A -85,B 0,C 180,E1 -8193.544,E2 -8193.544} C_VEL
LIN {X 0,Y 455.351,Z 529.374,A -85,B 0,C 180,E1 -8194.537,E2 -8194.537} C_VEL
LIN {X 0,Y 455.886,Z 518.274,A -85,B 0,C 180,E1 -8195.307,E2 -8195.307} C_VEL
LIN {X 0,Y 456.195,Z 507.092,A -85,B 0,C 180,E1 -8195.913,E2 -8195.913} C_VEL
LIN {X 0,Y 456.519,Z 494.417,A -85,B 0,C 180,E1 -8196.408,E2 -8196.408} C_VEL
LIN {X 0,Y 456.821,Z 480.979,A -85,B 0,C 180,E1 -8196.737,E2 -8196.737} C_VEL
LIN {X 0,Y 457.581,Z 393.227,A -85,B 0,C 180,E1 -8198.118,E2 -8198.118} C_VEL
LIN {X 0,Y 454.615,Z 378.81,A -85,B 0,C 180,E1 -8198.484,E2 -8198.484} C_VEL
LIN {X 0,Y 454.589,Z 371.139,A -85,B 0,C 180,E1 -8200.241,E2 -8200.241} C_VEL
LIN {X 0,Y 453.61,Z 364.985,A -85,B 0,C 180,E1 -8201.725,E2 -8201.725} C_VEL
LIN {X 0,Y 453.555,Z 364.984,A -85,B 0,C 180,E1 -8205.273,E2 -8205.273} C_VEL
LIN {X 0,Y 453.515,Z 364.992,A -85,B 0,C 180,E1 -8208.055,E2 -8208.055} C_VEL
LIN {X 0,Y 453.487,Z 364.995,A -85,B 0,C 180,E1 -8210.882,E2 -8210.882} C_VEL
LIN {X 0,Y 453.504,Z 364.993,A -85,B 0,C 180,E1 -8213.888,E2 -8213.888} C_VEL
LIN {X 0,Y 453.512,Z 364.992,A -85,B 0,C 180,E1 -8216.705,E2 -8216.705} C_VEL
LIN {X 0,Y 453.491,Z 364.995,A -85,B 0,C 180,E1 -8219.788,E2 -8219.788} C_VEL
LIN {X 0,Y 453.492,Z 364.994,A -85,B 0,C 180,E1 -8223.188,E2 -8223.188} C_VEL
LIN {X 0,Y 453.456,Z 365.002,A -85,B 0,C 180,E1 -8226.299,E2 -8226.299} C_VEL
LIN {X 0,Y 453.489,Z 364.995,A -85,B 0,C 180,E1 -8229.449,E2 -8229.449} C_VEL
LIN {X 0,Y 453.475,Z 365,A -85,B 0,C 180,E1 -8231.934,E2 -8231.934} C_VEL
LIN {X 0,Y 453.491,Z 364.995,A -85,B 0,C 180,E1 -8235.469,E2 -8235.469} C_VEL
LIN {X 0,Y 453.494,Z 364.997,A -85,B 0,C 180,E1 -8238.21,E2 -8238.21} C_VEL
LIN {X 0,Y 453.527,Z 364.99,A -85,B 0,C 180,E1 -8240.787,E2 -8240.787} C_VEL
LIN {X 0,Y 453.452,Z 365.003,A -85,B 0,C 180,E1 -8243.916,E2 -8243.916} C_VEL
LIN {X 0,Y 453.478,Z 364.997,A -85,B 0,C 180,E1 -8247.15,E2 -8247.15} C_VEL
LIN {X 0,Y 453.469,Z 364.999,A -85,B 0,C 180,E1 -8250.267,E2 -8250.267} C_VEL
LIN {X 0,Y 453.508,Z 364.994,A -85,B 0,C 180,E1 -8253.294,E2 -8253.294} C_VEL
LIN {X 0,Y 453.498,Z 364.995,A -85,B 0,C 180,E1 -8256.238,E2 -8256.238} C_VEL
LIN {X 0,Y 453.5,Z 364.995,A -85,B 0,C 180,E1 -8259.118,E2 -8259.118} C_VEL
LIN {X 0,Y 453.504,Z 364.995,A -85,B 0,C 180,E1 -8261.944,E2 -8261.944} C_VEL
LIN {X 0,Y 453.533,Z 364.992,A -85,B 0,C 180,E1 -8264.726,E2 -8264.726} C_VEL
LIN {X 0,Y 453.594,Z 364.984,A -85,B 0,C 180,E1 -8267.472,E2 -8267.472} C_VEL
LIN {X 0,Y 453.585,Z 364.984,A -85,B 0,C 180,E1 -8271.086,E2 -8271.086} C_VEL
LIN {X 0,Y 453.669,Z 364.974,A -85,B 0,C 180,E1 -8273.774,E2 -8273.774} C_VEL
LIN {X 0,Y 453.758,Z 364.963,A -85,B 0,C 180,E1 -8277.337,E2 -8277.337} C_VEL
LIN {X 0,Y 453.815,Z 364.955,A -85,B 0,C 180,E1 -8280,E2 -8280} C_VEL
LIN {X 0,Y 453.758,Z 364.964,A -85,B 0,C 180,E1 -8282.663,E2 -8282.663} C_VEL
LIN {X 0,Y 453.671,Z 364.974,A -85,B 0,C 180,E1 -8286.225,E2 -8286.225} C_VEL
LIN {X 0,Y 453.585,Z 364.984,A -85,B 0,C 180,E1 -8288.913,E2 -8288.913} C_VEL
LIN {X 0,Y 453.593,Z 364.985,A -85,B 0,C 180,E1 -8292.551,E2 -8292.551} C_VEL
LIN {X 0,Y 453.536,Z 364.992,A -85,B 0,C 180,E1 -8296.196,E2 -8296.196} C_VEL
LIN {X 0,Y 453.512,Z 364.993,A -85,B 0,C 180,E1 -8299.041,E2 -8299.041} C_VEL
LIN {X 0,Y 453.49,Z 364.996,A -85,B 0,C 180,E1 -8301.835,E2 -8301.835} C_VEL
LIN {X 0,Y 453.507,Z 364.994,A -85,B 0,C 180,E1 -8304.735,E2 -8304.735} C_VEL
LIN {X 0,Y 453.53,Z 364.992,A -85,B 0,C 180,E1 -8307.961,E2 -8307.961} C_VEL
LIN {X 0,Y 453.459,Z 364.999,A -85,B 0,C 180,E1 -8311.526,E2 -8311.526} C_VEL
LIN {X 0,Y 453.483,Z 364.996,A -85,B 0,C 180,E1 -8314.778,E2 -8314.778} C_VEL
LIN {X 0,Y 453.478,Z 364.999,A -85,B 0,C 180,E1 -8318.31,E2 -8318.31} C_VEL
LIN {X 0,Y 453.511,Z 364.992,A -85,B 0,C 180,E1 -8320.607,E2 -8320.607} C_VEL
LIN {X 0,Y 453.477,Z 364.996,A -85,B 0,C 180,E1 -8323.248,E2 -8323.248} C_VEL
LIN {X 0,Y 453.462,Z 365,A -85,B 0,C 180,E1 -8325.78,E2 -8325.78} C_VEL
LIN {X 0,Y 453.475,Z 364.999,A -85,B 0,C 180,E1 -8328.21,E2 -8328.21} C_VEL
LIN {X 0,Y 453.491,Z 364.993,A -85,B 0,C 180,E1 -8330.794,E2 -8330.794} C_VEL
LIN {X 0,Y 453.455,Z 365.004,A -85,B 0,C 180,E1 -8333.918,E2 -8333.918} C_VEL
LIN {X 0,Y 453.482,Z 364.994,A -85,B 0,C 180,E1 -8337.152,E2 -8337.152} C_VEL
LIN {X 0,Y 453.513,Z 364.997,A -85,B 0,C 180,E1 -8340.272,E2 -8340.272} C_VEL
LIN {X 0,Y 453.59,Z 365.175,A -85,B 0,C 180,E1 -8343.113,E2 -8343.113} C_VEL
LIN {X 0,Y 456.078,Z 378.052,A -85,B 0,C 180,E1 -8345.554,E2 -8345.554} C_VEL
LIN {X 0,Y 455.418,Z 393.5,A -85,B 0,C 180,E1 -8348.262,E2 -8348.262} C_VEL
LIN {X 0,Y 454.482,Z 413.659,A -85,B 0,C 180,E1 -8351.752,E2 -8351.752} C_VEL
LIN {X 0,Y 454.303,Z 418.353,A -85,B 0,C 180,E1 -8352.542,E2 -8352.542} C_VEL
LIN {X 0,Y 457.402,Z 439.991,A -85,B 0,C 180,E1 -8352.996,E2 -8352.996} C_VEL
LIN {X 0,Y 456.698,Z 526.846,A -85,B 0,C 180,E1 -8354.378,E2 -8354.378} C_VEL
LIN {X 0,Y 456.313,Z 540.155,A -85,B 0,C 180,E1 -8354.765,E2 -8354.765} C_VEL
LIN {X 0,Y 455.769,Z 552.92,A -85,B 0,C 180,E1 -8355.318,E2 -8355.318} C_VEL
LIN {X 0,Y 455.207,Z 565.055,A -85,B 0,C 180,E1 -8356.041,E2 -8356.041} C_VEL
LIN {X 0,Y 454.572,Z 577.315,A -85,B 0,C 180,E1 -8356.993,E2 -8356.993} C_VEL
LIN {X 0,Y 454.107,Z 588.071,A -85,B 0,C 180,E1 -8358.054,E2 -8358.054} C_VEL
LIN {X 0,Y 453.54,Z 598.053,A -85,B 0,C 180,E1 -8359.284,E2 -8359.284} C_VEL
LIN {X 0,Y 453.109,Z 606.84,A -85,B 0,C 180,E1 -8360.627,E2 -8360.627} C_VEL
LIN {X 0,Y 452.837,Z 613.846,A -85,B 0,C 180,E1 -8361.971,E2 -8361.971} C_VEL
LIN {X 0,Y 452.634,Z 619.457,A -85,B 0,C 180,E1 -8363.313,E2 -8363.313} C_VEL
LIN {X 0,Y 452.578,Z 623.861,A -85,B 0,C 180,E1 -8364.654,E2 -8364.654} C_VEL
LIN {X 0,Y 452.494,Z 626.186,A -85,B 0,C 180,E1 -8365.546,E2 -8365.546} C_VEL
LIN {X 0,Y 452.507,Z 628.081,A -85,B 0,C 180,E1 -8366.438,E2 -8366.438} C_VEL
LIN {X 0,Y 452.525,Z 629.51,A -85,B 0,C 180,E1 -8367.33,E2 -8367.33} C_VEL
LIN {X 0,Y 452.488,Z 631.145,A -85,B 0,C 180,E1 -8369.11,E2 -8369.11} C_VEL
LIN {X 0,Y 452.465,Z 631.377,A -85,B 0,C 180,E1 -8370,E2 -8370} C_VEL
LIN {X 0,Y 452.488,Z 631.18,A -85,B 0,C 180,E1 -8370.89,E2 -8370.89} C_VEL
LIN {X 0,Y 452.523,Z 629.591,A -85,B 0,C 180,E1 -8372.67,E2 -8372.67} C_VEL
LIN {X 0,Y 452.492,Z 628.202,A -85,B 0,C 180,E1 -8373.562,E2 -8373.562} C_VEL
LIN {X 0,Y 452.551,Z 625.277,A -85,B 0,C 180,E1 -8374.9,E2 -8374.9} C_VEL
LIN {X 0,Y 452.61,Z 620.797,A -85,B 0,C 180,E1 -8376.396,E2 -8376.396} C_VEL
LIN {X 0,Y 452.778,Z 616.232,A -85,B 0,C 180,E1 -8377.581,E2 -8377.581} C_VEL
LIN {X 0,Y 453.003,Z 609.849,A -85,B 0,C 180,E1 -8378.925,E2 -8378.925} C_VEL
LIN {X 0,Y 453.369,Z 601.877,A -85,B 0,C 180,E1 -8380.269,E2 -8380.269} C_VEL
LIN {X 0,Y 453.989,Z 591.987,A -85,B 0,C 180,E1 -8381.61,E2 -8381.61} C_VEL
LIN {X 0,Y 454.5,Z 582.605,A -85,B 0,C 180,E1 -8382.638,E2 -8382.638} C_VEL
LIN {X 0,Y 455.069,Z 571.462,A -85,B 0,C 180,E1 -8383.622,E2 -8383.622} C_VEL
LIN {X 0,Y 455.67,Z 560.342,A -85,B 0,C 180,E1 -8384.4,E2 -8384.4} C_VEL
LIN {X 0,Y 456.252,Z 547.977,A -85,B 0,C 180,E1 -8385.066,E2 -8385.066} C_VEL
LIN {X 0,Y 456.81,Z 534.827,A -85,B 0,C 180,E1 -8385.561,E2 -8385.561} C_VEL
LIN {X 0,Y 457.088,Z 522.178,A -85,B 0,C 180,E1 -8385.866,E2 -8385.866} C_VEL
LIN {X 0,Y 457.699,Z 439.125,A -85,B 0,C 180,E1 -8387.192,E2 -8387.192} C_VEL
LIN {X 0,Y 454.471,Z 417.884,A -85,B 0,C 180,E1 -8387.701,E2 -8387.701} C_VEL
LIN {X 0,Y 455.47,Z 397.643,A -85,B 0,C 180,E1 -8391.26,E2 -8391.26} C_VEL
LIN {X 0,Y 456.452,Z 380.523,A -85,B 0,C 180,E1 -8394.322,E2 -8394.322} C_VEL
LIN {X 0,Y 455.742,Z 375.249,A -85,B 0,C 180,E1 -8395.336,E2 -8395.336} C_VEL
LIN {X 0,Y 453.58,Z 364.987,A -85,B 0,C 180,E1 -8397.417,E2 -8397.417} C_VEL
LIN {X 0,Y 453.482,Z 364.993,A -85,B 0,C 180,E1 -8400.758,E2 -8400.758} C_VEL
LIN {X 0,Y 453.476,Z 365.001,A -85,B 0,C 180,E1 -8403.912,E2 -8403.912} C_VEL
LIN {X 0,Y 453.468,Z 364.997,A -85,B 0,C 180,E1 -8407.187,E2 -8407.187} C_VEL
LIN {X 0,Y 453.514,Z 364.992,A -85,B 0,C 180,E1 -8409.446,E2 -8409.446} C_VEL
LIN {X 0,Y 453.459,Z 364.995,A -85,B 0,C 180,E1 -8412.994,E2 -8412.994} C_VEL
LIN {X 0,Y 453.472,Z 364.998,A -85,B 0,C 180,E1 -8415.78,E2 -8415.78} C_VEL
LIN {X 0,Y 453.491,Z 364.992,A -85,B 0,C 180,E1 -8418.211,E2 -8418.211} C_VEL
LIN {X 0,Y 453.521,Z 364.987,A -85,B 0,C 180,E1 -8420.788,E2 -8420.788} C_VEL
LIN {X 0,Y 453.451,Z 365,A -85,B 0,C 180,E1 -8423.917,E2 -8423.917} C_VEL
LIN {X 0,Y 453.476,Z 364.997,A -85,B 0,C 180,E1 -8427.151,E2 -8427.151} C_VEL
LIN {X 0,Y 453.507,Z 364.99,A -85,B 0,C 180,E1 -8430.271,E2 -8430.271} C_VEL
LIN {X 0,Y 453.506,Z 364.991,A -85,B 0,C 180,E1 -8433.294,E2 -8433.294} C_VEL
LIN {X 0,Y 453.497,Z 364.985,A -85,B 0,C 180,E1 -8436.239,E2 -8436.239} C_VEL
LIN {X 0,Y 453.485,Z 364.999,A -85,B 0,C 180,E1 -8439.118,E2 -8439.118} C_VEL
LIN {X 0,Y 453.503,Z 364.991,A -85,B 0,C 180,E1 -8441.944,E2 -8441.944} C_VEL
LIN {X 0,Y 453.531,Z 364.988,A -85,B 0,C 180,E1 -8444.726,E2 -8444.726} C_VEL
LIN {X 0,Y 453.593,Z 364.983,A -85,B 0,C 180,E1 -8447.472,E2 -8447.472} C_VEL
LIN {X 0,Y 453.585,Z 364.987,A -85,B 0,C 180,E1 -8451.087,E2 -8451.087} C_VEL
LIN {X 0,Y 453.669,Z 364.966,A -85,B 0,C 180,E1 -8453.775,E2 -8453.775} C_VEL
LIN {X 0,Y 453.758,Z 364.96,A -85,B 0,C 180,E1 -8457.337,E2 -8457.337} C_VEL
LIN {X 0,Y 453.815,Z 364.951,A -85,B 0,C 180,E1 -8460,E2 -8460} C_VEL
LIN {X 0,Y 453.758,Z 364.964,A -85,B 0,C 180,E1 -8462.663,E2 -8462.663} C_VEL
LIN {X 0,Y 453.669,Z 364.972,A -85,B 0,C 180,E1 -8466.226,E2 -8466.226} C_VEL
LIN {X 0,Y 453.585,Z 364.985,A -85,B 0,C 180,E1 -8468.914,E2 -8468.914} C_VEL
LIN {X 0,Y 453.555,Z 364.987,A -85,B 0,C 180,E1 -8472.529,E2 -8472.529} C_VEL
LIN {X 0,Y 453.537,Z 364.99,A -85,B 0,C 180,E1 -8476.197,E2 -8476.197} C_VEL
LIN {X 0,Y 453.513,Z 364.991,A -85,B 0,C 180,E1 -8479.041,E2 -8479.041} C_VEL
LIN {X 0,Y 453.469,Z 364.994,A -85,B 0,C 180,E1 -8481.837,E2 -8481.837} C_VEL
LIN {X 0,Y 453.508,Z 364.987,A -85,B 0,C 180,E1 -8484.735,E2 -8484.735} C_VEL
LIN {X 0,Y 453.531,Z 364.984,A -85,B 0,C 180,E1 -8487.962,E2 -8487.962} C_VEL
LIN {X 0,Y 453.461,Z 364.995,A -85,B 0,C 180,E1 -8491.526,E2 -8491.526} C_VEL
LIN {X 0,Y 453.485,Z 364.995,A -85,B 0,C 180,E1 -8494.779,E2 -8494.779} C_VEL
LIN {X 0,Y 453.477,Z 365,A -85,B 0,C 180,E1 -8498.311,E2 -8498.311} C_VEL
LIN {X 0,Y 453.513,Z 364.994,A -85,B 0,C 180,E1 -8500.607,E2 -8500.607} C_VEL
LIN {X 0,Y 453.479,Z 364.995,A -85,B 0,C 180,E1 -8503.249,E2 -8503.249} C_VEL
LIN {X 0,Y 453.464,Z 365.002,A -85,B 0,C 180,E1 -8505.78,E2 -8505.78} C_VEL
LIN {X 0,Y 453.516,Z 364.995,A -85,B 0,C 180,E1 -8509.407,E2 -8509.407} C_VEL
LIN {X 0,Y 453.479,Z 364.999,A -85,B 0,C 180,E1 -8512.223,E2 -8512.223} C_VEL
LIN {X 0,Y 453.49,Z 364.997,A -85,B 0,C 180,E1 -8515.223,E2 -8515.223} C_VEL
LIN {X 0,Y 453.47,Z 365,A -85,B 0,C 180,E1 -8518.475,E2 -8518.475} C_VEL
LIN {X 0,Y 453.534,Z 365.026,A -85,B 0,C 180,E1 -8519.973,E2 -8519.973} C_VEL
LIN {X 0,Y 454.82,Z 372.082,A -85,B 0,C 180,E1 -8521.738,E2 -8521.738} C_VEL
LIN {X 0,Y 454.804,Z 379.069,A -85,B 0,C 180,E1 -8523.377,E2 -8523.377} C_VEL
LIN {X 0,Y 458.145,Z 394.414,A -85,B 0,C 180,E1 -8523.797,E2 -8523.797} C_VEL
LIN {X 0,Y 457.203,Z 486.266,A -85,B 0,C 180,E1 -8525.279,E2 -8525.279} C_VEL
LIN {X 0,Y 456.914,Z 498.495,A -85,B 0,C 180,E1 -8525.644,E2 -8525.644} C_VEL
LIN {X 0,Y 456.482,Z 511.616,A -85,B 0,C 180,E1 -8526.223,E2 -8526.223} C_VEL
LIN {X 0,Y 456.062,Z 522.302,A -85,B 0,C 180,E1 -8526.862,E2 -8526.862} C_VEL
LIN {X 0,Y 455.983,Z 524.587,A -85,B 0,C 180,E1 -8527.024,E2 -8527.024} C_VEL
LIN {X 0,Y 455.073,Z 529.728,A -85,B 0,C 180,E1 -8527.382,E2 -8527.382} C_VEL
LIN {X 0,Y 451.843,Z 537.844,A -85,B 0,C 180,E1 -8527.973,E2 -8527.973} C_VEL
LIN {X 0,Y 448.597,Z 545.523,A -85,B 0,C 180,E1 -8528.652,E2 -8528.652} C_VEL
LIN {X 0,Y 447.667,Z 549.905,A -85,B 0,C 180,E1 -8529.142,E2 -8529.142} C_VEL
LIN {X 0,Y 447.148,Z 558.471,A -85,B 0,C 180,E1 -8530.298,E2 -8530.298} C_VEL
LIN {X 0,Y 446.581,Z 566.613,A -85,B 0,C 180,E1 -8531.655,E2 -8531.655} C_VEL
LIN {X 0,Y 446.213,Z 573.369,A -85,B 0,C 180,E1 -8533.06,E2 -8533.06} C_VEL
LIN {X 0,Y 445.876,Z 578.711,A -85,B 0,C 180,E1 -8534.458,E2 -8534.458} C_VEL
LIN {X 0,Y 445.661,Z 582.828,A -85,B 0,C 180,E1 -8535.852,E2 -8535.852} C_VEL
LIN {X 0,Y 445.553,Z 585.848,A -85,B 0,C 180,E1 -8537.242,E2 -8537.242} C_VEL
LIN {X 0,Y 445.501,Z 587.302,A -85,B 0,C 180,E1 -8538.166,E2 -8538.166} C_VEL
LIN {X 0,Y 445.422,Z 588.319,A -85,B 0,C 180,E1 -8539.086,E2 -8539.086} C_VEL
LIN {X 0,Y 445.362,Z 589.177,A -85,B 0,C 180,E1 -8540.921,E2 -8540.921} C_VEL
LIN {X 0,Y 445.38,Z 588.979,A -85,B 0,C 180,E1 -8541.836,E2 -8541.836} C_VEL
LIN {X 0,Y 445.513,Z 587.391,A -85,B 0,C 180,E1 -8543.66,E2 -8543.66} C_VEL
LIN {X 0,Y 445.535,Z 586.015,A -85,B 0,C 180,E1 -8544.569,E2 -8544.569} C_VEL
LIN {X 0,Y 445.627,Z 583.121,A -85,B 0,C 180,E1 -8545.93,E2 -8545.93} C_VEL
LIN {X 0,Y 445.799,Z 579.205,A -85,B 0,C 180,E1 -8547.289,E2 -8547.289} C_VEL
LIN {X 0,Y 445.95,Z 574.178,A -85,B 0,C 180,E1 -8548.645,E2 -8548.645} C_VEL
LIN {X 0,Y 446.399,Z 567.831,A -85,B 0,C 180,E1 -8550,E2 -8550} C_VEL
LIN {X 0,Y 446.815,Z 559.944,A -85,B 0,C 180,E1 -8551.352,E2 -8551.352} C_VEL
LIN {X 0,Y 447.338,Z 550.155,A -85,B 0,C 180,E1 -8552.701,E2 -8552.701} C_VEL
LIN {X 0,Y 447.844,Z 539.897,A -85,B 0,C 180,E1 -8553.824,E2 -8553.824} C_VEL
LIN {X 0,Y 448.424,Z 529.737,A -85,B 0,C 180,E1 -8554.72,E2 -8554.72} C_VEL
LIN {X 0,Y 448.99,Z 518.638,A -85,B 0,C 180,E1 -8555.502,E2 -8555.502} C_VEL
LIN {X 0,Y 449.3,Z 507.466,A -85,B 0,C 180,E1 -8556.117,E2 -8556.117} C_VEL
LIN {X 0,Y 449.645,Z 494.81,A -85,B 0,C 180,E1 -8556.619,E2 -8556.619} C_VEL
LIN {X 0,Y 449.953,Z 481.412,A -85,B 0,C 180,E1 -8556.953,E2 -8556.953} C_VEL
LIN {X 0,Y 450.747,Z 394.37,A -85,B 0,C 180,E1 -8558.343,E2 -8558.343} C_VEL
LIN {X 0,Y 447.657,Z 379.122,A -85,B 0,C 180,E1 -8558.732,E2 -8558.732} C_VEL
LIN {X 0,Y 447.543,Z 371.934,A -85,B 0,C 180,E1 -8560.404,E2 -8560.404} C_VEL
LIN {X 0,Y 446.581,Z 365.861,A -85,B 0,C 180,E1 -8561.899,E2 -8561.899} C_VEL
LIN {X 0,Y 446.522,Z 365.861,A -85,B 0,C 180,E1 -8565.519,E2 -8565.519} C_VEL
LIN {X 0,Y 446.479,Z 365.866,A -85,B 0,C 180,E1 -8569.184,E2 -8569.184} C_VEL
LIN {X 0,Y 446.423,Z 365.878,A -85,B 0,C 180,E1 -8572.199,E2 -8572.199} C_VEL
LIN {X 0,Y 446.461,Z 365.869,A -85,B 0,C 180,E1 -8575.151,E2 -8575.151} C_VEL
LIN {X 0,Y 446.487,Z 365.871,A -85,B 0,C 180,E1 -8578.178,E2 -8578.178} C_VEL
LIN {X 0,Y 446.421,Z 365.874,A -85,B 0,C 180,E1 -8581.299,E2 -8581.299} C_VEL
LIN {X 0,Y 446.432,Z 365.876,A -85,B 0,C 180,E1 -8584.522,E2 -8584.522} C_VEL
LIN {X 0,Y 446.431,Z 365.878,A -85,B 0,C 180,E1 -8588.081,E2 -8588.081} C_VEL
LIN {X 0,Y 446.426,Z 365.875,A -85,B 0,C 180,E1 -8590.917,E2 -8590.917} C_VEL
LIN {X 0,Y 446.4,Z 365.88,A -85,B 0,C 180,E1 -8593.845,E2 -8593.845} C_VEL
LIN {X 0,Y 446.444,Z 365.874,A -85,B 0,C 180,E1 -8596.396,E2 -8596.396} C_VEL
LIN {X 0,Y 446.465,Z 365.872,A -85,B 0,C 180,E1 -8599.804,E2 -8599.804} C_VEL
LIN {X 0,Y 446.429,Z 365.878,A -85,B 0,C 180,E1 -8602.123,E2 -8602.123} C_VEL
LIN {X 0,Y 446.425,Z 365.876,A -85,B 0,C 180,E1 -8605.476,E2 -8605.476} C_VEL
LIN {X 0,Y 446.411,Z 365.877,A -85,B 0,C 180,E1 -8608.699,E2 -8608.699} C_VEL
LIN {X 0,Y 446.479,Z 365.872,A -85,B 0,C 180,E1 -8611.82,E2 -8611.82} C_VEL
LIN {X 0,Y 446.453,Z 365.873,A -85,B 0,C 180,E1 -8614.847,E2 -8614.847} C_VEL
LIN {X 0,Y 446.463,Z 365.871,A -85,B 0,C 180,E1 -8618.237,E2 -8618.237} C_VEL
LIN {X 0,Y 446.45,Z 365.874,A -85,B 0,C 180,E1 -8621.649,E2 -8621.649} C_VEL
LIN {X 0,Y 446.501,Z 365.867,A -85,B 0,C 180,E1 -8624.479,E2 -8624.479} C_VEL
LIN {X 0,Y 446.538,Z 365.862,A -85,B 0,C 180,E1 -8628.193,E2 -8628.193} C_VEL
LIN {X 0,Y 446.592,Z 365.856,A -85,B 0,C 180,E1 -8631.857,E2 -8631.857} C_VEL
LIN {X 0,Y 446.638,Z 365.851,A -85,B 0,C 180,E1 -8634.582,E2 -8634.582} C_VEL
LIN {X 0,Y 446.702,Z 365.842,A -85,B 0,C 180,E1 -8637.294,E2 -8637.294} C_VEL
LIN {X 0,Y 446.786,Z 365.831,A -85,B 0,C 180,E1 -8640,E2 -8640} C_VEL
LIN {X 0,Y 446.702,Z 365.842,A -85,B 0,C 180,E1 -8642.705,E2 -8642.705} C_VEL
LIN {X 0,Y 446.64,Z 365.851,A -85,B 0,C 180,E1 -8646.324,E2 -8646.324} C_VEL
LIN {X 0,Y 446.531,Z 365.862,A -85,B 0,C 180,E1 -8649.055,E2 -8649.055} C_VEL
LIN {X 0,Y 446.526,Z 365.864,A -85,B 0,C 180,E1 -8652.729,E2 -8652.729} C_VEL
LIN {X 0,Y 446.481,Z 365.871,A -85,B 0,C 180,E1 -8656.459,E2 -8656.459} C_VEL
LIN {X 0,Y 446.462,Z 365.871,A -85,B 0,C 180,E1 -8659.303,E2 -8659.303} C_VEL
LIN {X 0,Y 446.426,Z 365.878,A -85,B 0,C 180,E1 -8662.199,E2 -8662.199} C_VEL
LIN {X 0,Y 446.451,Z 365.872,A -85,B 0,C 180,E1 -8665.153,E2 -8665.153} C_VEL
LIN {X 0,Y 446.477,Z 365.872,A -85,B 0,C 180,E1 -8668.179,E2 -8668.179} C_VEL
LIN {X 0,Y 446.413,Z 365.877,A -85,B 0,C 180,E1 -8671.776,E2 -8671.776} C_VEL
LIN {X 0,Y 446.424,Z 365.876,A -85,B 0,C 180,E1 -8674.523,E2 -8674.523} C_VEL
LIN {X 0,Y 446.431,Z 365.879,A -85,B 0,C 180,E1 -8678.084,E2 -8678.084} C_VEL
LIN {X 0,Y 446.442,Z 365.872,A -85,B 0,C 180,E1 -8680.921,E2 -8680.921} C_VEL
LIN {X 0,Y 446.44,Z 365.875,A -85,B 0,C 180,E1 -8683.841,E2 -8683.841} C_VEL
LIN {X 0,Y 446.395,Z 365.879,A -85,B 0,C 180,E1 -8686.404,E2 -8686.404} C_VEL
LIN {X 0,Y 446.423,Z 365.874,A -85,B 0,C 180,E1 -8689.083,E2 -8689.083} C_VEL
LIN {X 0,Y 446.425,Z 365.878,A -85,B 0,C 180,E1 -8692.124,E2 -8692.124} C_VEL
LIN {X 0,Y 446.429,Z 365.875,A -85,B 0,C 180,E1 -8695.478,E2 -8695.478} C_VEL
LIN {X 0,Y 446.419,Z 365.874,A -85,B 0,C 180,E1 -8698.701,E2 -8698.701} C_VEL
LIN {X 0,Y 446.484,Z 365.873,A -85,B 0,C 180,E1 -8701.822,E2 -8701.822} C_VEL
LIN {X 0,Y 446.539,Z 366.004,A -85,B 0,C 180,E1 -8702.902,E2 -8702.902} C_VEL
LIN {X 0,Y 448.923,Z 378.051,A -85,B 0,C 180,E1 -8705.231,E2 -8705.231} C_VEL
LIN {X 0,Y 448.983,Z 383.554,A -85,B 0,C 180,E1 -8706.23,E2 -8706.23} C_VEL
LIN {X 0,Y 448.16,Z 399.741,A -85,B 0,C 180,E1 -8709.099,E2 -8709.099} C_VEL
LIN {X 0,Y 447.286,Z 417.901,A -85,B 0,C 180,E1 -8712.285,E2 -8712.285} C_VEL
LIN {X 0,Y 450.541,Z 441.397,A -85,B 0,C 180,E1 -8712.784,E2 -8712.784} C_VEL
LIN {X 0,Y 449.826,Z 526.614,A -85,B 0,C 180,E1 -8714.162,E2 -8714.162} C_VEL
LIN {X 0,Y 449.385,Z 539.889,A -85,B 0,C 180,E1 -8714.553,E2 -8714.553} C_VEL
LIN {X 0,Y 448.874,Z 552.075,A -85,B 0,C 180,E1 -8715.087,E2 -8715.087} C_VEL
LIN {X 0,Y 448.263,Z 564.367,A -85,B 0,C 180,E1 -8715.82,E2 -8715.82} C_VEL
LIN {X 0,Y 447.66,Z 575.854,A -85,B 0,C 180,E1 -8716.713,E2 -8716.713} C_VEL
LIN {X 0,Y 447.127,Z 586.487,A -85,B 0,C 180,E1 -8717.749,E2 -8717.749} C_VEL
LIN {X 0,Y 446.651,Z 595.907,A -85,B 0,C 180,E1 -8718.887,E2 -8718.887} C_VEL
LIN {X 0,Y 446.132,Z 605.01,A -85,B 0,C 180,E1 -8720.25,E2 -8720.25} C_VEL
LIN {X 0,Y 445.817,Z 612.347,A -85,B 0,C 180,E1 -8721.615,E2 -8721.615} C_VEL
LIN {X 0,Y 445.616,Z 617.304,A -85,B 0,C 180,E1 -8722.752,E2 -8722.752} C_VEL
LIN {X 0,Y 445.458,Z 621.657,A -85,B 0,C 180,E1 -8723.969,E2 -8723.969} C_VEL
LIN {X 0,Y 445.42,Z 625.803,A -85,B 0,C 180,E1 -8725.475,E2 -8725.475} C_VEL
LIN {X 0,Y 445.407,Z 627.707,A -85,B 0,C 180,E1 -8726.381,E2 -8726.381} C_VEL
LIN {X 0,Y 445.449,Z 629.152,A -85,B 0,C 180,E1 -8727.287,E2 -8727.287} C_VEL
LIN {X 0,Y 445.395,Z 630.8,A -85,B 0,C 180,E1 -8729.096,E2 -8729.096} C_VEL
LIN {X 0,Y 445.401,Z 631.042,A -85,B 0,C 180,E1 -8730,E2 -8730} C_VEL
LIN {X 0,Y 445.395,Z 630.857,A -85,B 0,C 180,E1 -8730.904,E2 -8730.904} C_VEL
LIN {X 0,Y 445.447,Z 629.282,A -85,B 0,C 180,E1 -8732.713,E2 -8732.713} C_VEL
LIN {X 0,Y 445.391,Z 627.9,A -85,B 0,C 180,E1 -8733.619,E2 -8733.619} C_VEL
LIN {X 0,Y 445.481,Z 624.992,A -85,B 0,C 180,E1 -8734.978,E2 -8734.978} C_VEL
LIN {X 0,Y 445.555,Z 619.643,A -85,B 0,C 180,E1 -8736.748,E2 -8736.748} C_VEL
LIN {X 0,Y 445.765,Z 614,A -85,B 0,C 180,E1 -8738.157,E2 -8738.157} C_VEL
LIN {X 0,Y 446.078,Z 607.163,A -85,B 0,C 180,E1 -8739.522,E2 -8739.522} C_VEL
LIN {X 0,Y 446.563,Z 598.67,A -85,B 0,C 180,E1 -8740.886,E2 -8740.886} C_VEL
LIN {X 0,Y 447.147,Z 589.948,A -85,B 0,C 180,E1 -8742.02,E2 -8742.02} C_VEL
LIN {X 0,Y 447.704,Z 579.128,A -85,B 0,C 180,E1 -8743.167,E2 -8743.167} C_VEL
LIN {X 0,Y 448.326,Z 568.595,A -85,B 0,C 180,E1 -8744.062,E2 -8744.062} C_VEL
LIN {X 0,Y 448.967,Z 556.713,A -85,B 0,C 180,E1 -8744.852,E2 -8744.852} C_VEL
LIN {X 0,Y 449.6,Z 544.372,A -85,B 0,C 180,E1 -8745.469,E2 -8745.469} C_VEL
LIN {X 0,Y 450.11,Z 531.71,A -85,B 0,C 180,E1 -8745.915,E2 -8745.915} C_VEL
LIN {X 0,Y 450.37,Z 516.722,A -85,B 0,C 180,E1 -8746.226,E2 -8746.226} C_VEL
LIN {X 0,Y 451.02,Z 440.203,A -85,B 0,C 180,E1 -8747.46,E2 -8747.46} C_VEL
LIN {X 0,Y 447.522,Z 417.564,A -85,B 0,C 180,E1 -8748.012,E2 -8748.012} C_VEL
LIN {X 0,Y 448.593,Z 397.517,A -85,B 0,C 180,E1 -8751.602,E2 -8751.602} C_VEL
LIN {X 0,Y 449.566,Z 381.86,A -85,B 0,C 180,E1 -8754.451,E2 -8754.451} C_VEL
LIN {X 0,Y 448.239,Z 373.85,A -85,B 0,C 180,E1 -8756.04,E2 -8756.04} C_VEL
LIN {X 0,Y 446.5,Z 365.869,A -85,B 0,C 180,E1 -8757.73,E2 -8757.73} C_VEL
LIN {X 0,Y 446.435,Z 365.875,A -85,B 0,C 180,E1 -8760.248,E2 -8760.248} C_VEL
LIN {X 0,Y 446.443,Z 365.874,A -85,B 0,C 180,E1 -8763.453,E2 -8763.453} C_VEL
LIN {X 0,Y 446.407,Z 365.877,A -85,B 0,C 180,E1 -8766.744,E2 -8766.744} C_VEL
LIN {X 0,Y 446.475,Z 365.87,A -85,B 0,C 180,E1 -8769.528,E2 -8769.528} C_VEL
LIN {X 0,Y 446.425,Z 365.872,A -85,B 0,C 180,E1 -8772.604,E2 -8772.604} C_VEL
LIN {X 0,Y 446.452,Z 365.868,A -85,B 0,C 180,E1 -8775.102,E2 -8775.102} C_VEL
LIN {X 0,Y 446.439,Z 365.868,A -85,B 0,C 180,E1 -8778.61,E2 -8778.61} C_VEL
LIN {X 0,Y 446.465,Z 365.867,A -85,B 0,C 180,E1 -8780.975,E2 -8780.975} C_VEL
LIN {X 0,Y 446.415,Z 365.873,A -85,B 0,C 180,E1 -8784.374,E2 -8784.374} C_VEL
LIN {X 0,Y 446.416,Z 365.88,A -85,B 0,C 180,E1 -8787.638,E2 -8787.638} C_VEL
LIN {X 0,Y 446.462,Z 365.868,A -85,B 0,C 180,E1 -8790.792,E2 -8790.792} C_VEL
LIN {X 0,Y 446.47,Z 365.859,A -85,B 0,C 180,E1 -8793.848,E2 -8793.848} C_VEL
LIN {X 0,Y 446.423,Z 365.868,A -85,B 0,C 180,E1 -8796.823,E2 -8796.823} C_VEL
LIN {X 0,Y 446.44,Z 365.871,A -85,B 0,C 180,E1 -8799.737,E2 -8799.737} C_VEL
LIN {X 0,Y 446.455,Z 365.87,A -85,B 0,C 180,E1 -8802.597,E2 -8802.597} C_VEL
LIN {X 0,Y 446.462,Z 365.871,A -85,B 0,C 180,E1 -8805.412,E2 -8805.412} C_VEL
LIN {X 0,Y 446.532,Z 365.859,A -85,B 0,C 180,E1 -8808.194,E2 -8808.194} C_VEL
LIN {X 0,Y 446.591,Z 365.852,A -85,B 0,C 180,E1 -8811.858,E2 -8811.858} C_VEL
LIN {X 0,Y 446.638,Z 365.844,A -85,B 0,C 180,E1 -8814.583,E2 -8814.583} C_VEL
LIN {X 0,Y 446.702,Z 365.839,A -85,B 0,C 180,E1 -8817.295,E2 -8817.295} C_VEL
LIN {X 0,Y 446.785,Z 365.826,A -85,B 0,C 180,E1 -8820,E2 -8820} C_VEL
LIN {X 0,Y 446.702,Z 365.842,A -85,B 0,C 180,E1 -8822.706,E2 -8822.706} C_VEL
LIN {X 0,Y 446.638,Z 365.849,A -85,B 0,C 180,E1 -8826.324,E2 -8826.324} C_VEL
LIN {X 0,Y 446.531,Z 365.862,A -85,B 0,C 180,E1 -8829.056,E2 -8829.056} C_VEL
LIN {X 0,Y 446.513,Z 365.864,A -85,B 0,C 180,E1 -8832.73,E2 -8832.73} C_VEL
LIN {X 0,Y 446.488,Z 365.868,A -85,B 0,C 180,E1 -8836.229,E2 -8836.229} C_VEL
LIN {X 0,Y 446.462,Z 365.868,A -85,B 0,C 180,E1 -8839.304,E2 -8839.304} C_VEL
LIN {X 0,Y 446.411,Z 365.877,A -85,B 0,C 180,E1 -8842.2,E2 -8842.2} C_VEL
LIN {X 0,Y 446.451,Z 365.863,A -85,B 0,C 180,E1 -8845.153,E2 -8845.153} C_VEL
LIN {X 0,Y 446.479,Z 365.865,A -85,B 0,C 180,E1 -8848.18,E2 -8848.18} C_VEL
LIN {X 0,Y 446.414,Z 365.874,A -85,B 0,C 180,E1 -8851.776,E2 -8851.776} C_VEL
LIN {X 0,Y 446.426,Z 365.877,A -85,B 0,C 180,E1 -8854.524,E2 -8854.524} C_VEL
LIN {X 0,Y 446.432,Z 365.88,A -85,B 0,C 180,E1 -8858.084,E2 -8858.084} C_VEL
LIN {X 0,Y 446.444,Z 365.873,A -85,B 0,C 180,E1 -8860.922,E2 -8860.922} C_VEL
LIN {X 0,Y 446.443,Z 365.877,A -85,B 0,C 180,E1 -8863.842,E2 -8863.842} C_VEL
LIN {X 0,Y 446.398,Z 365.881,A -85,B 0,C 180,E1 -8866.404,E2 -8866.404} C_VEL
LIN {X 0,Y 446.468,Z 365.876,A -85,B 0,C 180,E1 -8869.806,E2 -8869.806} C_VEL
LIN {X 0,Y 446.435,Z 365.877,A -85,B 0,C 180,E1 -8872.125,E2 -8872.125} C_VEL
LIN {X 0,Y 446.432,Z 365.876,A -85,B 0,C 180,E1 -8875.478,E2 -8875.478} C_VEL
LIN {X 0,Y 446.423,Z 365.878,A -85,B 0,C 180,E1 -8878.701,E2 -8878.701} C_VEL
LIN {X 0,Y 446.49,Z 366.02,A -85,B 0,C 180,E1 -8879.756,E2 -8879.756} C_VEL
LIN {X 0,Y 447.797,Z 372.914,A -85,B 0,C 180,E1 -8881.511,E2 -8881.511} C_VEL
LIN {X 0,Y 447.969,Z 377.781,A -85,B 0,C 180,E1 -8882.685,E2 -8882.685} C_VEL
LIN {X 0,Y 447.906,Z 379.46,A -85,B 0,C 180,E1 -8883.08,E2 -8883.08} C_VEL
LIN {X 0,Y 451.444,Z 395.372,A -85,B 0,C 180,E1 -8883.513,E2 -8883.513} C_VEL
LIN {X 0,Y 450.474,Z 485.948,A -85,B 0,C 180,E1 -8884.992,E2 -8884.992} C_VEL
LIN {X 0,Y 450.149,Z 498.797,A -85,B 0,C 180,E1 -8885.377,E2 -8885.377} C_VEL
LIN {X 0,Y 449.691,Z 511.921,A -85,B 0,C 180,E1 -8885.964,E2 -8885.964} C_VEL
LIN {X 0,Y 449.244,Z 522.61,A -85,B 0,C 180,E1 -8886.612,E2 -8886.612} C_VEL
LIN {X 0,Y 448.739,Z 533.426,A -85,B 0,C 180,E1 -8887.448,E2 -8887.448} C_VEL
LIN {X 0,Y 448.046,Z 544.225,A -85,B 0,C 180,E1 -8888.491,E2 -8888.491} C_VEL
LIN {X 0,Y 447.667,Z 549.905,A -85,B 0,C 180,E1 -8889.142,E2 -8889.142} C_VEL
LIN {X 0,Y 446.729,Z 554.176,A -85,B 0,C 180,E1 -8889.662,E2 -8889.662} C_VEL
LIN {X 0,Y 443.44,Z 560.73,A -85,B 0,C 180,E1 -8890.521,E2 -8890.521} C_VEL
LIN {X 0,Y 440.219,Z 566.744,A -85,B 0,C 180,E1 -8891.454,E2 -8891.454} C_VEL
LIN {X 0,Y 439.395,Z 570.013,A -85,B 0,C 180,E1 -8892.083,E2 -8892.083} C_VEL
LIN {X 0,Y 439.002,Z 576.792,A -85,B 0,C 180,E1 -8893.679,E2 -8893.679} C_VEL
LIN {X 0,Y 438.707,Z 581.587,A -85,B 0,C 180,E1 -8895.149,E2 -8895.149} C_VEL
LIN {X 0,Y 438.564,Z 583.993,A -85,B 0,C 180,E1 -8896.092,E2 -8896.092} C_VEL
LIN {X 0,Y 438.48,Z 585.953,A -85,B 0,C 180,E1 -8897.033,E2 -8897.033} C_VEL
LIN {X 0,Y 438.426,Z 587.485,A -85,B 0,C 180,E1 -8897.972,E2 -8897.972} C_VEL
LIN {X 0,Y 438.342,Z 588.552,A -85,B 0,C 180,E1 -8898.908,E2 -8898.908} C_VEL
LIN {X 0,Y 438.276,Z 589.492,A -85,B 0,C 180,E1 -8900.773,E2 -8900.773} C_VEL
LIN {X 0,Y 438.292,Z 589.372,A -85,B 0,C 180,E1 -8901.703,E2 -8901.703} C_VEL
LIN {X 0,Y 438.426,Z 587.868,A -85,B 0,C 180,E1 -8903.557,E2 -8903.557} C_VEL
LIN {X 0,Y 438.447,Z 586.537,A -85,B 0,C 180,E1 -8904.481,E2 -8904.481} C_VEL
LIN {X 0,Y 438.516,Z 583.726,A -85,B 0,C 180,E1 -8905.864,E2 -8905.864} C_VEL
LIN {X 0,Y 438.739,Z 579.896,A -85,B 0,C 180,E1 -8907.246,E2 -8907.246} C_VEL
LIN {X 0,Y 438.88,Z 574.968,A -85,B 0,C 180,E1 -8908.624,E2 -8908.624} C_VEL
LIN {X 0,Y 439.316,Z 568.762,A -85,B 0,C 180,E1 -8910,E2 -8910} C_VEL
LIN {X 0,Y 439.747,Z 561.021,A -85,B 0,C 180,E1 -8911.374,E2 -8911.374} C_VEL
LIN {X 0,Y 440.315,Z 551.377,A -85,B 0,C 180,E1 -8912.745,E2 -8912.745} C_VEL
LIN {X 0,Y 440.828,Z 541.394,A -85,B 0,C 180,E1 -8913.885,E2 -8913.885} C_VEL
LIN {X 0,Y 441.505,Z 530.07,A -85,B 0,C 180,E1 -8914.908,E2 -8914.908} C_VEL
LIN {X 0,Y 442.087,Z 518.969,A -85,B 0,C 180,E1 -8915.702,E2 -8915.702} C_VEL
LIN {X 0,Y 442.415,Z 507.792,A -85,B 0,C 180,E1 -8916.327,E2 -8916.327} C_VEL
LIN {X 0,Y 442.767,Z 495.133,A -85,B 0,C 180,E1 -8916.837,E2 -8916.837} C_VEL
LIN {X 0,Y 443.088,Z 481.726,A -85,B 0,C 180,E1 -8917.175,E2 -8917.175} C_VEL
LIN {X 0,Y 443.89,Z 395.228,A -85,B 0,C 180,E1 -8918.579,E2 -8918.579} C_VEL
LIN {X 0,Y 440.694,Z 379.509,A -85,B 0,C 180,E1 -8918.971,E2 -8918.971} C_VEL
LIN {X 0,Y 440.512,Z 372.726,A -85,B 0,C 180,E1 -8920.572,E2 -8920.572} C_VEL
LIN {X 0,Y 439.548,Z 366.737,A -85,B 0,C 180,E1 -8922.087,E2 -8922.087} C_VEL
LIN {X 0,Y 439.481,Z 366.742,A -85,B 0,C 180,E1 -8925.774,E2 -8925.774} C_VEL
LIN {X 0,Y 439.446,Z 366.742,A -85,B 0,C 180,E1 -8929.337,E2 -8929.337} C_VEL
LIN {X 0,Y 439.37,Z 366.756,A -85,B 0,C 180,E1 -8932.575,E2 -8932.575} C_VEL
LIN {X 0,Y 439.408,Z 366.748,A -85,B 0,C 180,E1 -8935.584,E2 -8935.584} C_VEL
LIN {X 0,Y 439.428,Z 366.747,A -85,B 0,C 180,E1 -8938.672,E2 -8938.672} C_VEL
LIN {X 0,Y 439.376,Z 366.754,A -85,B 0,C 180,E1 -8941.859,E2 -8941.859} C_VEL
LIN {X 0,Y 439.402,Z 366.749,A -85,B 0,C 180,E1 -8945.155,E2 -8945.155} C_VEL
LIN {X 0,Y 439.388,Z 366.752,A -85,B 0,C 180,E1 -8948.593,E2 -8948.593} C_VEL
LIN {X 0,Y 439.387,Z 366.751,A -85,B 0,C 180,E1 -8951.256,E2 -8951.256} C_VEL
LIN {X 0,Y 439.401,Z 366.75,A -85,B 0,C 180,E1 -8954.728,E2 -8954.728} C_VEL
LIN {X 0,Y 439.41,Z 366.75,A -85,B 0,C 180,E1 -8957.797,E2 -8957.797} C_VEL
LIN {X 0,Y 439.447,Z 366.747,A -85,B 0,C 180,E1 -8960.229,E2 -8960.229} C_VEL
LIN {X 0,Y 439.372,Z 366.755,A -85,B 0,C 180,E1 -8963.712,E2 -8963.712} C_VEL
LIN {X 0,Y 439.368,Z 366.755,A -85,B 0,C 180,E1 -8967.053,E2 -8967.053} C_VEL
LIN {X 0,Y 439.377,Z 366.754,A -85,B 0,C 180,E1 -8970.273,E2 -8970.273} C_VEL
LIN {X 0,Y 439.424,Z 366.748,A -85,B 0,C 180,E1 -8973.395,E2 -8973.395} C_VEL
LIN {X 0,Y 439.382,Z 366.753,A -85,B 0,C 180,E1 -8976.429,E2 -8976.429} C_VEL
LIN {X 0,Y 439.398,Z 366.751,A -85,B 0,C 180,E1 -8979.397,E2 -8979.397} C_VEL
LIN {X 0,Y 439.424,Z 366.748,A -85,B 0,C 180,E1 -8982.309,E2 -8982.309} C_VEL
LIN {X 0,Y 439.443,Z 366.745,A -85,B 0,C 180,E1 -8985.173,E2 -8985.173} C_VEL
LIN {X 0,Y 439.504,Z 366.739,A -85,B 0,C 180,E1 -8988.002,E2 -8988.002} C_VEL
LIN {X 0,Y 439.54,Z 366.735,A -85,B 0,C 180,E1 -8991.726,E2 -8991.726} C_VEL
LIN {X 0,Y 439.613,Z 366.726,A -85,B 0,C 180,E1 -8994.495,E2 -8994.495} C_VEL
LIN {X 0,Y 439.628,Z 366.723,A -85,B 0,C 180,E1 -8998.168,E2 -8998.168} C_VEL
LIN {X 0,Y 439.756,Z 366.707,A -85,B 0,C 180,E1 -9000,E2 -9000} C_VEL
LIN {X 0,Y 439.649,Z 366.721,A -85,B 0,C 180,E1 -9002.749,E2 -9002.749} C_VEL
LIN {X 0,Y 439.611,Z 366.727,A -85,B 0,C 180,E1 -9006.425,E2 -9006.425} C_VEL
LIN {X 0,Y 439.493,Z 366.739,A -85,B 0,C 180,E1 -9009.202,E2 -9009.202} C_VEL
LIN {X 0,Y 439.496,Z 366.739,A -85,B 0,C 180,E1 -9012.727,E2 -9012.727} C_VEL
LIN {X 0,Y 439.439,Z 366.749,A -85,B 0,C 180,E1 -9016.349,E2 -9016.349} C_VEL
LIN {X 0,Y 439.426,Z 366.747,A -85,B 0,C 180,E1 -9019.625,E2 -9019.625} C_VEL
LIN {X 0,Y 439.366,Z 366.756,A -85,B 0,C 180,E1 -9022.575,E2 -9022.575} C_VEL
LIN {X 0,Y 439.398,Z 366.751,A -85,B 0,C 180,E1 -9025.585,E2 -9025.585} C_VEL
LIN {X 0,Y 439.41,Z 366.749,A -85,B 0,C 180,E1 -9028.674,E2 -9028.674} C_VEL
LIN {X 0,Y 439.364,Z 366.758,A -85,B 0,C 180,E1 -9032.031,E2 -9032.031} C_VEL
LIN {X 0,Y 439.39,Z 366.751,A -85,B 0,C 180,E1 -9035.341,E2 -9035.341} C_VEL
LIN {X 0,Y 439.392,Z 366.751,A -85,B 0,C 180,E1 -9038.594,E2 -9038.594} C_VEL
LIN {X 0,Y 439.4,Z 366.75,A -85,B 0,C 180,E1 -9041.26,E2 -9041.26} C_VEL
LIN {X 0,Y 439.404,Z 366.749,A -85,B 0,C 180,E1 -9044.729,E2 -9044.729} C_VEL
LIN {X 0,Y 439.392,Z 366.754,A -85,B 0,C 180,E1 -9047.796,E2 -9047.796} C_VEL
LIN {X 0,Y 439.422,Z 366.749,A -85,B 0,C 180,E1 -9050.228,E2 -9050.228} C_VEL
LIN {X 0,Y 439.375,Z 366.755,A -85,B 0,C 180,E1 -9053.714,E2 -9053.714} C_VEL
LIN {X 0,Y 439.374,Z 366.751,A -85,B 0,C 180,E1 -9057.055,E2 -9057.055} C_VEL
LIN {X 0,Y 439.396,Z 366.756,A -85,B 0,C 180,E1 -9060.276,E2 -9060.276} C_VEL
LIN {X 0,Y 439.484,Z 366.883,A -85,B 0,C 180,E1 -9062.694,E2 -9062.694} C_VEL
LIN {X 0,Y 442.115,Z 380.613,A -85,B 0,C 180,E1 -9065.389,E2 -9065.389} C_VEL
LIN {X 0,Y 441.54,Z 393.848,A -85,B 0,C 180,E1 -9067.789,E2 -9067.789} C_VEL
LIN {X 0,Y 440.483,Z 413.992,A -85,B 0,C 180,E1 -9071.392,E2 -9071.392} C_VEL
LIN {X 0,Y 440.299,Z 417.542,A -85,B 0,C 180,E1 -9072.022,E2 -9072.022} C_VEL
LIN {X 0,Y 443.665,Z 441.123,A -85,B 0,C 180,E1 -9072.54,E2 -9072.54} C_VEL
LIN {X 0,Y 442.953,Z 526.281,A -85,B 0,C 180,E1 -9073.939,E2 -9073.939} C_VEL
LIN {X 0,Y 442.467,Z 539.555,A -85,B 0,C 180,E1 -9074.335,E2 -9074.335} C_VEL
LIN {X 0,Y 441.938,Z 552.315,A -85,B 0,C 180,E1 -9074.906,E2 -9074.906} C_VEL
LIN {X 0,Y 441.349,Z 563.643,A -85,B 0,C 180,E1 -9075.593,E2 -9075.593} C_VEL
LIN {X 0,Y 440.695,Z 575.428,A -85,B 0,C 180,E1 -9076.519,E2 -9076.519} C_VEL
LIN {X 0,Y 440.15,Z 585.898,A -85,B 0,C 180,E1 -9077.552,E2 -9077.552} C_VEL
LIN {X 0,Y 439.637,Z 595.382,A -85,B 0,C 180,E1 -9078.707,E2 -9078.707} C_VEL
LIN {X 0,Y 439.07,Z 604.518,A -85,B 0,C 180,E1 -9080.092,E2 -9080.092} C_VEL
LIN {X 0,Y 438.744,Z 611.886,A -85,B 0,C 180,E1 -9081.479,E2 -9081.479} C_VEL
LIN {X 0,Y 438.537,Z 616.869,A -85,B 0,C 180,E1 -9082.634,E2 -9082.634} C_VEL
LIN {X 0,Y 438.36,Z 621.671,A -85,B 0,C 180,E1 -9084.008,E2 -9084.008} C_VEL
LIN {X 0,Y 438.348,Z 625.414,A -85,B 0,C 180,E1 -9085.402,E2 -9085.402} C_VEL
LIN {X 0,Y 438.309,Z 627.326,A -85,B 0,C 180,E1 -9086.323,E2 -9086.323} C_VEL
LIN {X 0,Y 438.375,Z 628.79,A -85,B 0,C 180,E1 -9087.243,E2 -9087.243} C_VEL
LIN {X 0,Y 438.305,Z 630.454,A -85,B 0,C 180,E1 -9089.081,E2 -9089.081} C_VEL
LIN {X 0,Y 438.309,Z 630.704,A -85,B 0,C 180,E1 -9090,E2 -9090} C_VEL
LIN {X 0,Y 438.305,Z 630.535,A -85,B 0,C 180,E1 -9090.919,E2 -9090.919} C_VEL
LIN {X 0,Y 438.372,Z 628.978,A -85,B 0,C 180,E1 -9092.757,E2 -9092.757} C_VEL
LIN {X 0,Y 438.293,Z 627.603,A -85,B 0,C 180,E1 -9093.677,E2 -9093.677} C_VEL
LIN {X 0,Y 438.39,Z 624.713,A -85,B 0,C 180,E1 -9095.058,E2 -9095.058} C_VEL
LIN {X 0,Y 438.447,Z 620.792,A -85,B 0,C 180,E1 -9096.442,E2 -9096.442} C_VEL
LIN {X 0,Y 438.643,Z 615.75,A -85,B 0,C 180,E1 -9097.827,E2 -9097.827} C_VEL
LIN {X 0,Y 438.931,Z 609.43,A -85,B 0,C 180,E1 -9099.213,E2 -9099.213} C_VEL
LIN {X 0,Y 439.353,Z 601.534,A -85,B 0,C 180,E1 -9100.6,E2 -9100.6} C_VEL
LIN {X 0,Y 440.052,Z 591.72,A -85,B 0,C 180,E1 -9101.983,E2 -9101.983} C_VEL
LIN {X 0,Y 440.572,Z 582.282,A -85,B 0,C 180,E1 -9103.063,E2 -9103.063} C_VEL
LIN {X 0,Y 441.254,Z 571.468,A -85,B 0,C 180,E1 -9104.057,E2 -9104.057} C_VEL
LIN {X 0,Y 441.938,Z 560.524,A -85,B 0,C 180,E1 -9104.858,E2 -9104.858} C_VEL
LIN {X 0,Y 442.584,Z 548.436,A -85,B 0,C 180,E1 -9105.543,E2 -9105.543} C_VEL
LIN {X 0,Y 443.19,Z 535.966,A -85,B 0,C 180,E1 -9106.052,E2 -9106.052} C_VEL
LIN {X 0,Y 443.559,Z 523.005,A -85,B 0,C 180,E1 -9106.393,E2 -9106.393} C_VEL
LIN {X 0,Y 444.27,Z 440.695,A -85,B 0,C 180,E1 -9107.753,E2 -9107.753} C_VEL
LIN {X 0,Y 440.607,Z 417.273,A -85,B 0,C 180,E1 -9108.332,E2 -9108.332} C_VEL
LIN {X 0,Y 441.663,Z 398.717,A -85,B 0,C 180,E1 -9111.713,E2 -9111.713} C_VEL
LIN {X 0,Y 442.651,Z 382.469,A -85,B 0,C 180,E1 -9114.727,E2 -9114.727} C_VEL
LIN {X 0,Y 440.77,Z 372.538,A -85,B 0,C 180,E1 -9116.759,E2 -9116.759} C_VEL
LIN {X 0,Y 439.484,Z 366.742,A -85,B 0,C 180,E1 -9118.014,E2 -9118.014} C_VEL
LIN {X 0,Y 439.365,Z 366.751,A -85,B 0,C 180,E1 -9120.787,E2 -9120.787} C_VEL
LIN {X 0,Y 439.386,Z 366.756,A -85,B 0,C 180,E1 -9124.043,E2 -9124.043} C_VEL
LIN {X 0,Y 439.355,Z 366.755,A -85,B 0,C 180,E1 -9126.888,E2 -9126.888} C_VEL
LIN {X 0,Y 439.41,Z 366.751,A -85,B 0,C 180,E1 -9129.85,E2 -9129.85} C_VEL
LIN {X 0,Y 439.378,Z 366.749,A -85,B 0,C 180,E1 -9132.626,E2 -9132.626} C_VEL
LIN {X 0,Y 439.398,Z 366.75,A -85,B 0,C 180,E1 -9136.033,E2 -9136.033} C_VEL
LIN {X 0,Y 439.395,Z 366.747,A -85,B 0,C 180,E1 -9139.021,E2 -9139.021} C_VEL
LIN {X 0,Y 439.384,Z 366.754,A -85,B 0,C 180,E1 -9141.604,E2 -9141.604} C_VEL
LIN {X 0,Y 439.395,Z 366.748,A -85,B 0,C 180,E1 -9144.844,E2 -9144.844} C_VEL
LIN {X 0,Y 439.368,Z 366.753,A -85,B 0,C 180,E1 -9148.139,E2 -9148.139} C_VEL
LIN {X 0,Y 439.418,Z 366.751,A -85,B 0,C 180,E1 -9151.327,E2 -9151.327} C_VEL
LIN {X 0,Y 439.398,Z 366.738,A -85,B 0,C 180,E1 -9154.415,E2 -9154.415} C_VEL
LIN {X 0,Y 439.359,Z 366.756,A -85,B 0,C 180,E1 -9157.424,E2 -9157.424} C_VEL
LIN {X 0,Y 439.433,Z 366.743,A -85,B 0,C 180,E1 -9160.662,E2 -9160.662} C_VEL
LIN {X 0,Y 439.454,Z 366.739,A -85,B 0,C 180,E1 -9164.224,E2 -9164.224} C_VEL
LIN {X 0,Y 439.5,Z 366.735,A -85,B 0,C 180,E1 -9168.002,E2 -9168.002} C_VEL
LIN {X 0,Y 439.539,Z 366.731,A -85,B 0,C 180,E1 -9171.726,E2 -9171.726} C_VEL
LIN {X 0,Y 439.613,Z 366.719,A -85,B 0,C 180,E1 -9174.496,E2 -9174.496} C_VEL
LIN {X 0,Y 439.628,Z 366.718,A -85,B 0,C 180,E1 -9178.168,E2 -9178.168} C_VEL
LIN {X 0,Y 439.756,Z 366.702,A -85,B 0,C 180,E1 -9180,E2 -9180} C_VEL
LIN {X 0,Y 439.649,Z 366.719,A -85,B 0,C 180,E1 -9182.749,E2 -9182.749} C_VEL
LIN {X 0,Y 439.61,Z 366.726,A -85,B 0,C 180,E1 -9186.426,E2 -9186.426} C_VEL
LIN {X 0,Y 439.493,Z 366.738,A -85,B 0,C 180,E1 -9189.202,E2 -9189.202} C_VEL
LIN {X 0,Y 439.458,Z 366.743,A -85,B 0,C 180,E1 -9192.938,E2 -9192.938} C_VEL
LIN {X 0,Y 439.439,Z 366.747,A -85,B 0,C 180,E1 -9196.349,E2 -9196.349} C_VEL
LIN {X 0,Y 439.395,Z 366.749,A -85,B 0,C 180,E1 -9199.627,E2 -9199.627} C_VEL
LIN {X 0,Y 439.358,Z 366.759,A -85,B 0,C 180,E1 -9202.576,E2 -9202.576} C_VEL
LIN {X 0,Y 439.399,Z 366.741,A -85,B 0,C 180,E1 -9205.586,E2 -9205.586} C_VEL
LIN {X 0,Y 439.412,Z 366.75,A -85,B 0,C 180,E1 -9208.674,E2 -9208.674} C_VEL
LIN {X 0,Y 439.365,Z 366.755,A -85,B 0,C 180,E1 -9212.031,E2 -9212.031} C_VEL
LIN {X 0,Y 439.392,Z 366.75,A -85,B 0,C 180,E1 -9215.342,E2 -9215.342} C_VEL
LIN {X 0,Y 439.392,Z 366.751,A -85,B 0,C 180,E1 -9218.595,E2 -9218.595} C_VEL
LIN {X 0,Y 439.402,Z 366.751,A -85,B 0,C 180,E1 -9221.26,E2 -9221.26} C_VEL
LIN {X 0,Y 439.407,Z 366.752,A -85,B 0,C 180,E1 -9224.729,E2 -9224.729} C_VEL
LIN {X 0,Y 439.396,Z 366.758,A -85,B 0,C 180,E1 -9227.797,E2 -9227.797} C_VEL
LIN {X 0,Y 439.451,Z 366.747,A -85,B 0,C 180,E1 -9230.231,E2 -9230.231} C_VEL
LIN {X 0,Y 439.378,Z 366.755,A -85,B 0,C 180,E1 -9233.714,E2 -9233.714} C_VEL
LIN {X 0,Y 439.374,Z 366.754,A -85,B 0,C 180,E1 -9237.055,E2 -9237.055} C_VEL
LIN {X 0,Y 439.45,Z 366.834,A -85,B 0,C 180,E1 -9239.48,E2 -9239.48} C_VEL
LIN {X 0,Y 441,Z 375.435,A -85,B 0,C 180,E1 -9241.699,E2 -9241.699} C_VEL
LIN {X 0,Y 441.052,Z 380.02,A -85,B 0,C 180,E1 -9242.762,E2 -9242.762} C_VEL
LIN {X 0,Y 444.761,Z 396.215,A -85,B 0,C 180,E1 -9243.216,E2 -9243.216} C_VEL
LIN {X 0,Y 443.75,Z 486.483,A -85,B 0,C 180,E1 -9244.715,E2 -9244.715} C_VEL
LIN {X 0,Y 443.399,Z 498.37,A -85,B 0,C 180,E1 -9245.07,E2 -9245.07} C_VEL
LIN {X 0,Y 442.975,Z 511.116,A -85,B 0,C 180,E1 -9245.639,E2 -9245.639} C_VEL
LIN {X 0,Y 442.437,Z 522.955,A -85,B 0,C 180,E1 -9246.354,E2 -9246.354} C_VEL
LIN {X 0,Y 441.794,Z 535.066,A -85,B 0,C 180,E1 -9247.319,E2 -9247.319} C_VEL
LIN {X 0,Y 441.083,Z 545.653,A -85,B 0,C 180,E1 -9248.38,E2 -9248.38} C_VEL
LIN {X 0,Y 440.509,Z 554.333,A -85,B 0,C 180,E1 -9249.452,E2 -9249.452} C_VEL
LIN {X 0,Y 439.946,Z 561.952,A -85,B 0,C 180,E1 -9250.59,E2 -9250.59} C_VEL
LIN {X 0,Y 439.395,Z 570.013,A -85,B 0,C 180,E1 -9252.083,E2 -9252.083} C_VEL
LIN {X 0,Y 438.588,Z 573.098,A -85,B 0,C 180,E1 -9252.735,E2 -9252.735} C_VEL
LIN {X 0,Y 435.452,Z 577.702,A -85,B 0,C 180,E1 -9253.813,E2 -9253.813} C_VEL
LIN {X 0,Y 432.328,Z 581.644,A -85,B 0,C 180,E1 -9254.946,E2 -9254.946} C_VEL
LIN {X 0,Y 431.553,Z 583.604,A -85,B 0,C 180,E1 -9255.677,E2 -9255.677} C_VEL
LIN {X 0,Y 431.418,Z 586.064,A -85,B 0,C 180,E1 -9256.817,E2 -9256.817} C_VEL
LIN {X 0,Y 431.342,Z 587.765,A -85,B 0,C 180,E1 -9257.853,E2 -9257.853} C_VEL
LIN {X 0,Y 431.216,Z 589.491,A -85,B 0,C 180,E1 -9259.672,E2 -9259.672} C_VEL
LIN {X 0,Y 431.218,Z 589.736,A -85,B 0,C 180,E1 -9261.566,E2 -9261.566} C_VEL
LIN {X 0,Y 431.251,Z 589.25,A -85,B 0,C 180,E1 -9262.509,E2 -9262.509} C_VEL
LIN {X 0,Y 431.355,Z 588.098,A -85,B 0,C 180,E1 -9263.655,E2 -9263.655} C_VEL
LIN {X 0,Y 431.353,Z 585.367,A -85,B 0,C 180,E1 -9265.327,E2 -9265.327} C_VEL
LIN {X 0,Y 431.59,Z 581.965,A -85,B 0,C 180,E1 -9266.733,E2 -9266.733} C_VEL
LIN {X 0,Y 431.689,Z 577.517,A -85,B 0,C 180,E1 -9268.134,E2 -9268.134} C_VEL
LIN {X 0,Y 432.171,Z 570.751,A -85,B 0,C 180,E1 -9269.767,E2 -9269.767} C_VEL
LIN {X 0,Y 432.591,Z 563.434,A -85,B 0,C 180,E1 -9271.164,E2 -9271.164} C_VEL
LIN {X 0,Y 433.201,Z 554.335,A -85,B 0,C 180,E1 -9272.557,E2 -9272.557} C_VEL
LIN {X 0,Y 433.746,Z 543.861,A -85,B 0,C 180,E1 -9273.832,E2 -9273.832} C_VEL
LIN {X 0,Y 434.398,Z 533.175,A -85,B 0,C 180,E1 -9274.872,E2 -9274.872} C_VEL
LIN {X 0,Y 434.973,Z 522.769,A -85,B 0,C 180,E1 -9275.679,E2 -9275.679} C_VEL
LIN {X 0,Y 435.438,Z 510.311,A -85,B 0,C 180,E1 -9276.429,E2 -9276.429} C_VEL
LIN {X 0,Y 435.852,Z 497.127,A -85,B 0,C 180,E1 -9277.004,E2 -9277.004} C_VEL
LIN {X 0,Y 436.136,Z 484.939,A -85,B 0,C 180,E1 -9277.348,E2 -9277.348} C_VEL
LIN {X 0,Y 437.045,Z 396.115,A -85,B 0,C 180,E1 -9278.819,E2 -9278.819} C_VEL
LIN {X 0,Y 433.744,Z 379.833,A -85,B 0,C 180,E1 -9279.23,E2 -9279.23} C_VEL
LIN {X 0,Y 433.469,Z 373.516,A -85,B 0,C 180,E1 -9280.746,E2 -9280.746} C_VEL
LIN {X 0,Y 432.511,Z 367.614,A -85,B 0,C 180,E1 -9282.25,E2 -9282.25} C_VEL
LIN {X 0,Y 432.448,Z 367.62,A -85,B 0,C 180,E1 -9286.038,E2 -9286.038} C_VEL
LIN {X 0,Y 432.391,Z 367.621,A -85,B 0,C 180,E1 -9289.485,E2 -9289.485} C_VEL
LIN {X 0,Y 432.324,Z 367.631,A -85,B 0,C 180,E1 -9292.963,E2 -9292.963} C_VEL
LIN {X 0,Y 432.367,Z 367.627,A -85,B 0,C 180,E1 -9296.032,E2 -9296.032} C_VEL
LIN {X 0,Y 432.355,Z 367.627,A -85,B 0,C 180,E1 -9299.186,E2 -9299.186} C_VEL
LIN {X 0,Y 432.327,Z 367.635,A -85,B 0,C 180,E1 -9302.292,E2 -9302.292} C_VEL
LIN {X 0,Y 432.342,Z 367.63,A -85,B 0,C 180,E1 -9304.676,E2 -9304.676} C_VEL
LIN {X 0,Y 432.347,Z 367.633,A -85,B 0,C 180,E1 -9308.148,E2 -9308.148} C_VEL
LIN {X 0,Y 432.331,Z 367.63,A -85,B 0,C 180,E1 -9311.601,E2 -9311.601} C_VEL
LIN {X 0,Y 432.332,Z 367.633,A -85,B 0,C 180,E1 -9314.346,E2 -9314.346} C_VEL
LIN {X 0,Y 432.364,Z 367.627,A -85,B 0,C 180,E1 -9317.008,E2 -9317.008} C_VEL
LIN {X 0,Y 432.355,Z 367.629,A -85,B 0,C 180,E1 -9319.816,E2 -9319.816} C_VEL
LIN {X 0,Y 432.312,Z 367.633,A -85,B 0,C 180,E1 -9323.022,E2 -9323.022} C_VEL
LIN {X 0,Y 432.355,Z 367.632,A -85,B 0,C 180,E1 -9325.996,E2 -9325.996} C_VEL
LIN {X 0,Y 432.342,Z 367.63,A -85,B 0,C 180,E1 -9329.489,E2 -9329.489} C_VEL
LIN {X 0,Y 432.387,Z 367.625,A -85,B 0,C 180,E1 -9332.927,E2 -9332.927} C_VEL
LIN {X 0,Y 432.366,Z 367.629,A -85,B 0,C 180,E1 -9336.023,E2 -9336.023} C_VEL
LIN {X 0,Y 432.36,Z 367.627,A -85,B 0,C 180,E1 -9339.046,E2 -9339.046} C_VEL
LIN {X 0,Y 432.371,Z 367.628,A -85,B 0,C 180,E1 -9342.01,E2 -9342.01} C_VEL
LIN {X 0,Y 432.39,Z 367.624,A -85,B 0,C 180,E1 -9344.926,E2 -9344.926} C_VEL
LIN {X 0,Y 432.476,Z 367.615,A -85,B 0,C 180,E1 -9347.804,E2 -9347.804} C_VEL
LIN {X 0,Y 432.484,Z 367.614,A -85,B 0,C 180,E1 -9351.59,E2 -9351.59} C_VEL
LIN {X 0,Y 432.59,Z 367.6,A -85,B 0,C 180,E1 -9354.406,E2 -9354.406} C_VEL
LIN {X 0,Y 432.598,Z 367.599,A -85,B 0,C 180,E1 -9358.138,E2 -9358.138} C_VEL
LIN {X 0,Y 432.726,Z 367.583,A -85,B 0,C 180,E1 -9360,E2 -9360} C_VEL
LIN {X 0,Y 432.599,Z 367.598,A -85,B 0,C 180,E1 -9362.793,E2 -9362.793} C_VEL
LIN {X 0,Y 432.565,Z 367.604,A -85,B 0,C 180,E1 -9366.53,E2 -9366.53} C_VEL
LIN {X 0,Y 432.437,Z 367.618,A -85,B 0,C 180,E1 -9369.353,E2 -9369.353} C_VEL
LIN {X 0,Y 432.437,Z 367.618,A -85,B 0,C 180,E1 -9372.812,E2 -9372.812} C_VEL
LIN {X 0,Y 432.404,Z 367.624,A -85,B 0,C 180,E1 -9376.479,E2 -9376.479} C_VEL
LIN {X 0,Y 432.371,Z 367.627,A -85,B 0,C 180,E1 -9379.959,E2 -9379.959} C_VEL
LIN {X 0,Y 432.317,Z 367.632,A -85,B 0,C 180,E1 -9382.964,E2 -9382.964} C_VEL
LIN {X 0,Y 432.357,Z 367.63,A -85,B 0,C 180,E1 -9386.033,E2 -9386.033} C_VEL
LIN {X 0,Y 432.336,Z 367.63,A -85,B 0,C 180,E1 -9389.188,E2 -9389.188} C_VEL
LIN {X 0,Y 432.316,Z 367.634,A -85,B 0,C 180,E1 -9392.443,E2 -9392.443} C_VEL
LIN {X 0,Y 432.34,Z 367.63,A -85,B 0,C 180,E1 -9395.633,E2 -9395.633} C_VEL
LIN {X 0,Y 432.354,Z 367.627,A -85,B 0,C 180,E1 -9398.718,E2 -9398.718} C_VEL
LIN {X 0,Y 432.369,Z 367.628,A -85,B 0,C 180,E1 -9401.793,E2 -9401.793} C_VEL
LIN {X 0,Y 432.374,Z 367.626,A -85,B 0,C 180,E1 -9404.342,E2 -9404.342} C_VEL
LIN {X 0,Y 432.33,Z 367.633,A -85,B 0,C 180,E1 -9408.204,E2 -9408.204} C_VEL
LIN {X 0,Y 432.344,Z 367.628,A -85,B 0,C 180,E1 -9411.285,E2 -9411.285} C_VEL
LIN {X 0,Y 432.343,Z 367.629,A -85,B 0,C 180,E1 -9414.369,E2 -9414.369} C_VEL
LIN {X 0,Y 432.327,Z 367.632,A -85,B 0,C 180,E1 -9417.558,E2 -9417.558} C_VEL
LIN {X 0,Y 432.394,Z 367.626,A -85,B 0,C 180,E1 -9419.745,E2 -9419.745} C_VEL
LIN {X 0,Y 432.423,Z 367.693,A -85,B 0,C 180,E1 -9422.473,E2 -9422.473} C_VEL
LIN {X 0,Y 435.094,Z 381.166,A -85,B 0,C 180,E1 -9425.168,E2 -9425.168} C_VEL
LIN {X 0,Y 434.916,Z 388.07,A -85,B 0,C 180,E1 -9426.451,E2 -9426.451} C_VEL
LIN {X 0,Y 433.903,Z 405.698,A -85,B 0,C 180,E1 -9429.67,E2 -9429.67} C_VEL
LIN {X 0,Y 433.329,Z 417.375,A -85,B 0,C 180,E1 -9431.769,E2 -9431.769} C_VEL
LIN {X 0,Y 436.869,Z 443.081,A -85,B 0,C 180,E1 -9432.332,E2 -9432.332} C_VEL
LIN {X 0,Y 436.09,Z 525.857,A -85,B 0,C 180,E1 -9433.709,E2 -9433.709} C_VEL
LIN {X 0,Y 435.571,Z 539.159,A -85,B 0,C 180,E1 -9434.11,E2 -9434.11} C_VEL
LIN {X 0,Y 435.072,Z 551.375,A -85,B 0,C 180,E1 -9434.662,E2 -9434.662} C_VEL
LIN {X 0,Y 434.42,Z 562.87,A -85,B 0,C 180,E1 -9435.358,E2 -9435.358} C_VEL
LIN {X 0,Y 433.778,Z 574.173,A -85,B 0,C 180,E1 -9436.247,E2 -9436.247} C_VEL
LIN {X 0,Y 433.167,Z 585.284,A -85,B 0,C 180,E1 -9437.348,E2 -9437.348} C_VEL
LIN {X 0,Y 432.605,Z 594.832,A -85,B 0,C 180,E1 -9438.521,E2 -9438.521} C_VEL
LIN {X 0,Y 432.025,Z 604.012,A -85,B 0,C 180,E1 -9439.929,E2 -9439.929} C_VEL
LIN {X 0,Y 431.689,Z 611.413,A -85,B 0,C 180,E1 -9441.339,E2 -9441.339} C_VEL
LIN {X 0,Y 431.418,Z 618.189,A -85,B 0,C 180,E1 -9442.982,E2 -9442.982} C_VEL
LIN {X 0,Y 431.281,Z 622.658,A -85,B 0,C 180,E1 -9444.389,E2 -9444.389} C_VEL
LIN {X 0,Y 431.28,Z 625.018,A -85,B 0,C 180,E1 -9445.327,E2 -9445.327} C_VEL
LIN {X 0,Y 431.214,Z 626.939,A -85,B 0,C 180,E1 -9446.262,E2 -9446.262} C_VEL
LIN {X 0,Y 431.302,Z 628.424,A -85,B 0,C 180,E1 -9447.198,E2 -9447.198} C_VEL
LIN {X 0,Y 431.219,Z 630.107,A -85,B 0,C 180,E1 -9449.066,E2 -9449.066} C_VEL
LIN {X 0,Y 431.22,Z 630.365,A -85,B 0,C 180,E1 -9450,E2 -9450} C_VEL
LIN {X 0,Y 431.219,Z 630.215,A -85,B 0,C 180,E1 -9450.934,E2 -9450.934} C_VEL
LIN {X 0,Y 431.28,Z 628.676,A -85,B 0,C 180,E1 -9452.802,E2 -9452.802} C_VEL
LIN {X 0,Y 431.199,Z 627.311,A -85,B 0,C 180,E1 -9453.738,E2 -9453.738} C_VEL
LIN {X 0,Y 431.301,Z 624.441,A -85,B 0,C 180,E1 -9455.142,E2 -9455.142} C_VEL
LIN {X 0,Y 431.375,Z 620.543,A -85,B 0,C 180,E1 -9456.548,E2 -9456.548} C_VEL
LIN {X 0,Y 431.562,Z 615.525,A -85,B 0,C 180,E1 -9457.956,E2 -9457.956} C_VEL
LIN {X 0,Y 431.883,Z 609.236,A -85,B 0,C 180,E1 -9459.365,E2 -9459.365} C_VEL
LIN {X 0,Y 432.362,Z 601.389,A -85,B 0,C 180,E1 -9460.773,E2 -9460.773} C_VEL
LIN {X 0,Y 433.1,Z 591.618,A -85,B 0,C 180,E1 -9462.178,E2 -9462.178} C_VEL
LIN {X 0,Y 433.687,Z 581.511,A -85,B 0,C 180,E1 -9463.351,E2 -9463.351} C_VEL
LIN {X 0,Y 434.454,Z 570.093,A -85,B 0,C 180,E1 -9464.401,E2 -9464.401} C_VEL
LIN {X 0,Y 435.165,Z 558.908,A -85,B 0,C 180,E1 -9465.215,E2 -9465.215} C_VEL
LIN {X 0,Y 435.907,Z 546.384,A -85,B 0,C 180,E1 -9465.907,E2 -9465.907} C_VEL
LIN {X 0,Y 436.512,Z 533.009,A -85,B 0,C 180,E1 -9466.425,E2 -9466.425} C_VEL
LIN {X 0,Y 436.84,Z 519.878,A -85,B 0,C 180,E1 -9466.743,E2 -9466.743} C_VEL
LIN {X 0,Y 437.641,Z 441.812,A -85,B 0,C 180,E1 -9468.041,E2 -9468.041} C_VEL
LIN {X 0,Y 433.684,Z 416.952,A -85,B 0,C 180,E1 -9468.668,E2 -9468.668} C_VEL
LIN {X 0,Y 434.805,Z 398.612,A -85,B 0,C 180,E1 -9472.073,E2 -9472.073} C_VEL
LIN {X 0,Y 435.753,Z 384.205,A -85,B 0,C 180,E1 -9474.792,E2 -9474.792} C_VEL
LIN {X 0,Y 433.963,Z 374.506,A -85,B 0,C 180,E1 -9476.809,E2 -9476.809} C_VEL
LIN {X 0,Y 432.411,Z 367.621,A -85,B 0,C 180,E1 -9478.337,E2 -9478.337} C_VEL
LIN {X 0,Y 432.329,Z 367.628,A -85,B 0,C 180,E1 -9481.345,E2 -9481.345} C_VEL
LIN {X 0,Y 432.339,Z 367.631,A -85,B 0,C 180,E1 -9484.676,E2 -9484.676} C_VEL
LIN {X 0,Y 432.345,Z 367.631,A -85,B 0,C 180,E1 -9488.148,E2 -9488.148} C_VEL
LIN {X 0,Y 432.329,Z 367.632,A -85,B 0,C 180,E1 -9491.601,E2 -9491.601} C_VEL
LIN {X 0,Y 432.329,Z 367.628,A -85,B 0,C 180,E1 -9494.347,E2 -9494.347} C_VEL
LIN {X 0,Y 432.361,Z 367.623,A -85,B 0,C 180,E1 -9497.008,E2 -9497.008} C_VEL
LIN {X 0,Y 432.352,Z 367.629,A -85,B 0,C 180,E1 -9499.816,E2 -9499.816} C_VEL
LIN {X 0,Y 432.311,Z 367.63,A -85,B 0,C 180,E1 -9503.022,E2 -9503.022} C_VEL
LIN {X 0,Y 432.353,Z 367.628,A -85,B 0,C 180,E1 -9505.996,E2 -9505.996} C_VEL
LIN {X 0,Y 432.388,Z 367.624,A -85,B 0,C 180,E1 -9509.744,E2 -9509.744} C_VEL
LIN {X 0,Y 432.393,Z 367.618,A -85,B 0,C 180,E1 -9513.372,E2 -9513.372} C_VEL
LIN {X 0,Y 432.364,Z 367.618,A -85,B 0,C 180,E1 -9516.023,E2 -9516.023} C_VEL
LIN {X 0,Y 432.346,Z 367.631,A -85,B 0,C 180,E1 -9519.046,E2 -9519.046} C_VEL
LIN {X 0,Y 432.369,Z 367.624,A -85,B 0,C 180,E1 -9522.011,E2 -9522.011} C_VEL
LIN {X 0,Y 432.387,Z 367.623,A -85,B 0,C 180,E1 -9524.926,E2 -9524.926} C_VEL
LIN {X 0,Y 432.473,Z 367.611,A -85,B 0,C 180,E1 -9527.804,E2 -9527.804} C_VEL
LIN {X 0,Y 432.484,Z 367.611,A -85,B 0,C 180,E1 -9531.59,E2 -9531.59} C_VEL
LIN {X 0,Y 432.589,Z 367.593,A -85,B 0,C 180,E1 -9534.406,E2 -9534.406} C_VEL
LIN {X 0,Y 432.598,Z 367.594,A -85,B 0,C 180,E1 -9538.138,E2 -9538.138} C_VEL
LIN {X 0,Y 432.726,Z 367.578,A -85,B 0,C 180,E1 -9540,E2 -9540} C_VEL
LIN {X 0,Y 432.598,Z 367.597,A -85,B 0,C 180,E1 -9542.794,E2 -9542.794} C_VEL
LIN {X 0,Y 432.564,Z 367.605,A -85,B 0,C 180,E1 -9546.531,E2 -9546.531} C_VEL
LIN {X 0,Y 432.436,Z 367.616,A -85,B 0,C 180,E1 -9549.354,E2 -9549.354} C_VEL
LIN {X 0,Y 432.423,Z 367.619,A -85,B 0,C 180,E1 -9552.804,E2 -9552.804} C_VEL
LIN {X 0,Y 432.405,Z 367.622,A -85,B 0,C 180,E1 -9556.48,E2 -9556.48} C_VEL
LIN {X 0,Y 432.332,Z 367.631,A -85,B 0,C 180,E1 -9559.961,E2 -9559.961} C_VEL
LIN {X 0,Y 432.312,Z 367.632,A -85,B 0,C 180,E1 -9562.965,E2 -9562.965} C_VEL
LIN {X 0,Y 432.358,Z 367.617,A -85,B 0,C 180,E1 -9566.033,E2 -9566.033} C_VEL
LIN {X 0,Y 432.337,Z 367.628,A -85,B 0,C 180,E1 -9569.188,E2 -9569.188} C_VEL
LIN {X 0,Y 432.318,Z 367.635,A -85,B 0,C 180,E1 -9572.444,E2 -9572.444} C_VEL
LIN {X 0,Y 432.341,Z 367.63,A -85,B 0,C 180,E1 -9575.633,E2 -9575.633} C_VEL
LIN {X 0,Y 432.354,Z 367.627,A -85,B 0,C 180,E1 -9578.718,E2 -9578.718} C_VEL
LIN {X 0,Y 432.371,Z 367.628,A -85,B 0,C 180,E1 -9581.793,E2 -9581.793} C_VEL
LIN {X 0,Y 432.376,Z 367.631,A -85,B 0,C 180,E1 -9584.342,E2 -9584.342} C_VEL
LIN {X 0,Y 432.366,Z 367.63,A -85,B 0,C 180,E1 -9588.394,E2 -9588.394} C_VEL
LIN {X 0,Y 432.354,Z 367.632,A -85,B 0,C 180,E1 -9591.853,E2 -9591.853} C_VEL
LIN {X 0,Y 432.342,Z 367.631,A -85,B 0,C 180,E1 -9595.324,E2 -9595.324} C_VEL
LIN {X 0,Y 432.415,Z 367.766,A -85,B 0,C 180,E1 -9599.227,E2 -9599.227} C_VEL
LIN {X 0,Y 434.034,Z 376.538,A -85,B 0,C 180,E1 -9601.526,E2 -9601.526} C_VEL
LIN {X 0,Y 434.145,Z 380.117,A -85,B 0,C 180,E1 -9602.411,E2 -9602.411} C_VEL
LIN {X 0,Y 438.086,Z 397.089,A -85,B 0,C 180,E1 -9602.909,E2 -9602.909} C_VEL
LIN {X 0,Y 437.021,Z 486.95,A -85,B 0,C 180,E1 -9604.426,E2 -9604.426} C_VEL
LIN {X 0,Y 436.66,Z 498.793,A -85,B 0,C 180,E1 -9604.786,E2 -9604.786} C_VEL
LIN {X 0,Y 436.216,Z 511.513,A -85,B 0,C 180,E1 -9605.363,E2 -9605.363} C_VEL
LIN {X 0,Y 435.643,Z 523.334,A -85,B 0,C 180,E1 -9606.089,E2 -9606.089} C_VEL
LIN {X 0,Y 435.066,Z 534.273,A -85,B 0,C 180,E1 -9606.964,E2 -9606.964} C_VEL
LIN {X 0,Y 434.301,Z 544.915,A -85,B 0,C 180,E1 -9608.025,E2 -9608.025} C_VEL
LIN {X 0,Y 433.658,Z 553.773,A -85,B 0,C 180,E1 -9609.113,E2 -9609.113} C_VEL
LIN {X 0,Y 433.004,Z 562.356,A -85,B 0,C 180,E1 -9610.4,E2 -9610.4} C_VEL
LIN {X 0,Y 432.451,Z 569.715,A -85,B 0,C 180,E1 -9611.77,E2 -9611.77} C_VEL
LIN {X 0,Y 432.01,Z 576.777,A -85,B 0,C 180,E1 -9613.436,E2 -9613.436} C_VEL
LIN {X 0,Y 431.699,Z 581.578,A -85,B 0,C 180,E1 -9614.902,E2 -9614.902} C_VEL
LIN {X 0,Y 431.553,Z 583.604,A -85,B 0,C 180,E1 -9615.677,E2 -9615.677} C_VEL
LIN {X 0,Y 430.81,Z 585.368,A -85,B 0,C 180,E1 -9616.42,E2 -9616.42} C_VEL
LIN {X 0,Y 427.828,Z 587.762,A -85,B 0,C 180,E1 -9617.642,E2 -9617.642} C_VEL
LIN {X 0,Y 425.319,Z 589.1,A -85,B 0,C 180,E1 -9618.644,E2 -9618.644} C_VEL
LIN {X 0,Y 424.216,Z 589.728,A -85,B 0,C 180,E1 -9619.427,E2 -9619.427} C_VEL
LIN {X 0,Y 424.112,Z 589.839,A -85,B 0,C 180,E1 -9619.694,E2 -9619.694} C_VEL
LIN {X 0,Y 424.122,Z 590.09,A -85,B 0,C 180,E1 -9621.423,E2 -9621.423} C_VEL
LIN {X 0,Y 424.162,Z 589.671,A -85,B 0,C 180,E1 -9622.383,E2 -9622.383} C_VEL
LIN {X 0,Y 424.263,Z 588.416,A -85,B 0,C 180,E1 -9623.679,E2 -9623.679} C_VEL
LIN {X 0,Y 424.273,Z 585.919,A -85,B 0,C 180,E1 -9625.249,E2 -9625.249} C_VEL
LIN {X 0,Y 424.504,Z 582.601,A -85,B 0,C 180,E1 -9626.678,E2 -9626.678} C_VEL
LIN {X 0,Y 424.617,Z 578.241,A -85,B 0,C 180,E1 -9628.103,E2 -9628.103} C_VEL
LIN {X 0,Y 424.97,Z 572.689,A -85,B 0,C 180,E1 -9629.526,E2 -9629.526} C_VEL
LIN {X 0,Y 425.458,Z 565.757,A -85,B 0,C 180,E1 -9630.946,E2 -9630.946} C_VEL
LIN {X 0,Y 426.048,Z 557.091,A -85,B 0,C 180,E1 -9632.363,E2 -9632.363} C_VEL
LIN {X 0,Y 426.545,Z 548.248,A -85,B 0,C 180,E1 -9633.542,E2 -9633.542} C_VEL
LIN {X 0,Y 427.133,Z 538.524,A -85,B 0,C 180,E1 -9634.601,E2 -9634.601} C_VEL
LIN {X 0,Y 427.786,Z 527.787,A -85,B 0,C 180,E1 -9635.539,E2 -9635.539} C_VEL
LIN {X 0,Y 428.389,Z 515.773,A -85,B 0,C 180,E1 -9636.358,E2 -9636.358} C_VEL
LIN {X 0,Y 428.794,Z 503.259,A -85,B 0,C 180,E1 -9637.002,E2 -9637.002} C_VEL
LIN {X 0,Y 429.149,Z 490.925,A -85,B 0,C 180,E1 -9637.439,E2 -9637.439} C_VEL
LIN {X 0,Y 429.459,Z 475.243,A -85,B 0,C 180,E1 -9637.759,E2 -9637.759} C_VEL
LIN {X 0,Y 430.232,Z 397.223,A -85,B 0,C 180,E1 -9639.06,E2 -9639.06} C_VEL
LIN {X 0,Y 426.78,Z 380.1,A -85,B 0,C 180,E1 -9639.508,E2 -9639.508} C_VEL
LIN {X 0,Y 426.415,Z 374.305,A -85,B 0,C 180,E1 -9640.926,E2 -9640.926} C_VEL
LIN {X 0,Y 425.44,Z 368.494,A -85,B 0,C 180,E1 -9642.442,E2 -9642.442} C_VEL
LIN {X 0,Y 425.404,Z 368.498,A -85,B 0,C 180,E1 -9646.311,E2 -9646.311} C_VEL
LIN {X 0,Y 425.333,Z 368.5,A -85,B 0,C 180,E1 -9649.635,E2 -9649.635} C_VEL
LIN {X 0,Y 425.311,Z 368.503,A -85,B 0,C 180,E1 -9653.364,E2 -9653.364} C_VEL
LIN {X 0,Y 425.351,Z 368.5,A -85,B 0,C 180,E1 -9656.844,E2 -9656.844} C_VEL
LIN {X 0,Y 425.32,Z 368.503,A -85,B 0,C 180,E1 -9659.716,E2 -9659.716} C_VEL
LIN {X 0,Y 425.283,Z 368.508,A -85,B 0,C 180,E1 -9663.047,E2 -9663.047} C_VEL
LIN {X 0,Y 425.285,Z 368.51,A -85,B 0,C 180,E1 -9665.928,E2 -9665.928} C_VEL
LIN {X 0,Y 425.299,Z 368.506,A -85,B 0,C 180,E1 -9669.043,E2 -9669.043} C_VEL
LIN {X 0,Y 425.273,Z 368.51,A -85,B 0,C 180,E1 -9672.652,E2 -9672.652} C_VEL
LIN {X 0,Y 425.332,Z 368.506,A -85,B 0,C 180,E1 -9676.053,E2 -9676.053} C_VEL
LIN {X 0,Y 425.307,Z 368.506,A -85,B 0,C 180,E1 -9678.625,E2 -9678.625} C_VEL
LIN {X 0,Y 425.32,Z 368.504,A -85,B 0,C 180,E1 -9681.103,E2 -9681.103} C_VEL
LIN {X 0,Y 425.296,Z 368.508,A -85,B 0,C 180,E1 -9684.663,E2 -9684.663} C_VEL
LIN {X 0,Y 425.26,Z 368.515,A -85,B 0,C 180,E1 -9688.072,E2 -9688.072} C_VEL
LIN {X 0,Y 425.325,Z 368.503,A -85,B 0,C 180,E1 -9691.367,E2 -9691.367} C_VEL
LIN {X 0,Y 425.29,Z 368.509,A -85,B 0,C 180,E1 -9694.554,E2 -9694.554} C_VEL
LIN {X 0,Y 425.313,Z 368.507,A -85,B 0,C 180,E1 -9697.719,E2 -9697.719} C_VEL
LIN {X 0,Y 425.358,Z 368.501,A -85,B 0,C 180,E1 -9700.703,E2 -9700.703} C_VEL
LIN {X 0,Y 425.381,Z 368.498,A -85,B 0,C 180,E1 -9703.688,E2 -9703.688} C_VEL
LIN {X 0,Y 425.424,Z 368.493,A -85,B 0,C 180,E1 -9707.598,E2 -9707.598} C_VEL
LIN {X 0,Y 425.435,Z 368.491,A -85,B 0,C 180,E1 -9711.449,E2 -9711.449} C_VEL
LIN {X 0,Y 425.546,Z 368.478,A -85,B 0,C 180,E1 -9714.313,E2 -9714.313} C_VEL
LIN {X 0,Y 425.567,Z 368.475,A -85,B 0,C 180,E1 -9718.107,E2 -9718.107} C_VEL
LIN {X 0,Y 425.696,Z 368.459,A -85,B 0,C 180,E1 -9720,E2 -9720} C_VEL
LIN {X 0,Y 425.551,Z 368.476,A -85,B 0,C 180,E1 -9722.84,E2 -9722.84} C_VEL
LIN {X 0,Y 425.523,Z 368.48,A -85,B 0,C 180,E1 -9726.639,E2 -9726.639} C_VEL
LIN {X 0,Y 425.396,Z 368.496,A -85,B 0,C 180,E1 -9729.509,E2 -9729.509} C_VEL
LIN {X 0,Y 425.396,Z 368.495,A -85,B 0,C 180,E1 -9732.911,E2 -9732.911} C_VEL
LIN {X 0,Y 425.353,Z 368.501,A -85,B 0,C 180,E1 -9736.605,E2 -9736.605} C_VEL
LIN {X 0,Y 425.354,Z 368.501,A -85,B 0,C 180,E1 -9739.649,E2 -9739.649} C_VEL
LIN {X 0,Y 425.302,Z 368.507,A -85,B 0,C 180,E1 -9743.365,E2 -9743.365} C_VEL
LIN {X 0,Y 425.341,Z 368.501,A -85,B 0,C 180,E1 -9746.845,E2 -9746.845} C_VEL
LIN {X 0,Y 425.284,Z 368.51,A -85,B 0,C 180,E1 -9749.72,E2 -9749.72} C_VEL
LIN {X 0,Y 425.276,Z 368.509,A -85,B 0,C 180,E1 -9753.049,E2 -9753.049} C_VEL
LIN {X 0,Y 425.279,Z 368.512,A -85,B 0,C 180,E1 -9755.93,E2 -9755.93} C_VEL
LIN {X 0,Y 425.307,Z 368.505,A -85,B 0,C 180,E1 -9759.046,E2 -9759.046} C_VEL
LIN {X 0,Y 425.327,Z 368.502,A -85,B 0,C 180,E1 -9762.647,E2 -9762.647} C_VEL
LIN {X 0,Y 425.29,Z 368.507,A -85,B 0,C 180,E1 -9765.282,E2 -9765.282} C_VEL
LIN {X 0,Y 425.27,Z 368.509,A -85,B 0,C 180,E1 -9768.622,E2 -9768.622} C_VEL
LIN {X 0,Y 425.306,Z 368.504,A -85,B 0,C 180,E1 -9771.103,E2 -9771.103} C_VEL
LIN {X 0,Y 425.298,Z 368.505,A -85,B 0,C 180,E1 -9774.665,E2 -9774.665} C_VEL
LIN {X 0,Y 425.271,Z 368.512,A -85,B 0,C 180,E1 -9778.074,E2 -9778.074} C_VEL
LIN {X 0,Y 425.337,Z 368.504,A -85,B 0,C 180,E1 -9781.369,E2 -9781.369} C_VEL
LIN {X 0,Y 425.366,Z 368.504,A -85,B 0,C 180,E1 -9782.244,E2 -9782.244} C_VEL
LIN {X 0,Y 428.041,Z 381.98,A -85,B 0,C 180,E1 -9784.99,E2 -9784.99} C_VEL
LIN {X 0,Y 428.085,Z 387.409,A -85,B 0,C 180,E1 -9786.026,E2 -9786.026} C_VEL
LIN {X 0,Y 427.016,Z 404.897,A -85,B 0,C 180,E1 -9789.277,E2 -9789.277} C_VEL
LIN {X 0,Y 426.352,Z 417.089,A -85,B 0,C 180,E1 -9791.5,E2 -9791.5} C_VEL
LIN {X 0,Y 429.993,Z 442.871,A -85,B 0,C 180,E1 -9792.078,E2 -9792.078} C_VEL
LIN {X 0,Y 429.199,Z 525.332,A -85,B 0,C 180,E1 -9793.471,E2 -9793.471} C_VEL
LIN {X 0,Y 428.67,Z 538.705,A -85,B 0,C 180,E1 -9793.878,E2 -9793.878} C_VEL
LIN {X 0,Y 428.144,Z 551.527,A -85,B 0,C 180,E1 -9794.469,E2 -9794.469} C_VEL
LIN {X 0,Y 427.404,Z 563.691,A -85,B 0,C 180,E1 -9795.234,E2 -9795.234} C_VEL
LIN {X 0,Y 426.72,Z 575.673,A -85,B 0,C 180,E1 -9796.22,E2 -9796.22} C_VEL
LIN {X 0,Y 426.127,Z 585.73,A -85,B 0,C 180,E1 -9797.257,E2 -9797.257} C_VEL
LIN {X 0,Y 425.603,Z 594.261,A -85,B 0,C 180,E1 -9798.33,E2 -9798.33} C_VEL
LIN {X 0,Y 424.97,Z 603.492,A -85,B 0,C 180,E1 -9799.76,E2 -9799.76} C_VEL
LIN {X 0,Y 424.632,Z 610.928,A -85,B 0,C 180,E1 -9801.194,E2 -9801.194} C_VEL
LIN {X 0,Y 424.341,Z 617.748,A -85,B 0,C 180,E1 -9802.865,E2 -9802.865} C_VEL
LIN {X 0,Y 424.189,Z 622.242,A -85,B 0,C 180,E1 -9804.295,E2 -9804.295} C_VEL
LIN {X 0,Y 424.21,Z 624.616,A -85,B 0,C 180,E1 -9805.248,E2 -9805.248} C_VEL
LIN {X 0,Y 424.123,Z 626.548,A -85,B 0,C 180,E1 -9806.2,E2 -9806.2} C_VEL
LIN {X 0,Y 424.211,Z 628.054,A -85,B 0,C 180,E1 -9807.151,E2 -9807.151} C_VEL
LIN {X 0,Y 424.166,Z 629.102,A -85,B 0,C 180,E1 -9808.101,E2 -9808.101} C_VEL
LIN {X 0,Y 424.135,Z 630.026,A -85,B 0,C 180,E1 -9810,E2 -9810} C_VEL
LIN {X 0,Y 424.135,Z 629.895,A -85,B 0,C 180,E1 -9810.949,E2 -9810.949} C_VEL
LIN {X 0,Y 424.165,Z 629.332,A -85,B 0,C 180,E1 -9811.899,E2 -9811.899} C_VEL
LIN {X 0,Y 424.176,Z 628.377,A -85,B 0,C 180,E1 -9812.849,E2 -9812.849} C_VEL
LIN {X 0,Y 424.109,Z 627.023,A -85,B 0,C 180,E1 -9813.801,E2 -9813.801} C_VEL
LIN {X 0,Y 424.213,Z 624.175,A -85,B 0,C 180,E1 -9815.228,E2 -9815.228} C_VEL
LIN {X 0,Y 424.299,Z 620.301,A -85,B 0,C 180,E1 -9816.658,E2 -9816.658} C_VEL
LIN {X 0,Y 424.508,Z 615.31,A -85,B 0,C 180,E1 -9818.089,E2 -9818.089} C_VEL
LIN {X 0,Y 424.827,Z 609.051,A -85,B 0,C 180,E1 -9819.522,E2 -9819.522} C_VEL
LIN {X 0,Y 425.365,Z 601.258,A -85,B 0,C 180,E1 -9820.953,E2 -9820.953} C_VEL
LIN {X 0,Y 426.156,Z 591.533,A -85,B 0,C 180,E1 -9822.38,E2 -9822.38} C_VEL
LIN {X 0,Y 426.71,Z 582.247,A -85,B 0,C 180,E1 -9823.49,E2 -9823.49} C_VEL
LIN {X 0,Y 427.495,Z 571.593,A -85,B 0,C 180,E1 -9824.519,E2 -9824.519} C_VEL
LIN {X 0,Y 428.318,Z 559.088,A -85,B 0,C 180,E1 -9825.464,E2 -9825.464} C_VEL
LIN {X 0,Y 429.114,Z 546.787,A -85,B 0,C 180,E1 -9826.166,E2 -9826.166} C_VEL
LIN {X 0,Y 429.741,Z 533.756,A -85,B 0,C 180,E1 -9826.691,E2 -9826.691} C_VEL
LIN {X 0,Y 430.132,Z 519.837,A -85,B 0,C 180,E1 -9827.042,E2 -9827.042} C_VEL
LIN {X 0,Y 430.924,Z 442.4,A -85,B 0,C 180,E1 -9828.354,E2 -9828.354} C_VEL
LIN {X 0,Y 427.374,Z 419.995,A -85,B 0,C 180,E1 -9828.926,E2 -9828.926} C_VEL
LIN {X 0,Y 426.797,Z 416.496,A -85,B 0,C 180,E1 -9829.042,E2 -9829.042} C_VEL
LIN {X 0,Y 427.951,Z 398.517,A -85,B 0,C 180,E1 -9832.446,E2 -9832.446} C_VEL
LIN {X 0,Y 428.824,Z 386.745,A -85,B 0,C 180,E1 -9834.703,E2 -9834.703} C_VEL
LIN {X 0,Y 428.144,Z 381.197,A -85,B 0,C 180,E1 -9835.848,E2 -9835.848} C_VEL
LIN {X 0,Y 425.654,Z 369.768,A -85,B 0,C 180,E1 -9838.339,E2 -9838.339} C_VEL
LIN {X 0,Y 425.337,Z 368.502,A -85,B 0,C 180,E1 -9838.631,E2 -9838.631} C_VEL
LIN {X 0,Y 425.271,Z 368.513,A -85,B 0,C 180,E1 -9841.926,E2 -9841.926} C_VEL
LIN {X 0,Y 425.298,Z 368.508,A -85,B 0,C 180,E1 -9845.335,E2 -9845.335} C_VEL
LIN {X 0,Y 425.3,Z 368.505,A -85,B 0,C 180,E1 -9849.044,E2 -9849.044} C_VEL
LIN {X 0,Y 425.271,Z 368.507,A -85,B 0,C 180,E1 -9852.652,E2 -9852.652} C_VEL
LIN {X 0,Y 425.33,Z 368.502,A -85,B 0,C 180,E1 -9856.053,E2 -9856.053} C_VEL
LIN {X 0,Y 425.304,Z 368.501,A -85,B 0,C 180,E1 -9858.625,E2 -9858.625} C_VEL
LIN {X 0,Y 425.316,Z 368.502,A -85,B 0,C 180,E1 -9861.103,E2 -9861.103} C_VEL
LIN {X 0,Y 425.294,Z 368.504,A -85,B 0,C 180,E1 -9864.664,E2 -9864.664} C_VEL
LIN {X 0,Y 425.259,Z 368.511,A -85,B 0,C 180,E1 -9868.073,E2 -9868.073} C_VEL
LIN {X 0,Y 425.331,Z 368.506,A -85,B 0,C 180,E1 -9871.368,E2 -9871.368} C_VEL
LIN {X 0,Y 425.288,Z 368.495,A -85,B 0,C 180,E1 -9874.554,E2 -9874.554} C_VEL
LIN {X 0,Y 425.28,Z 368.51,A -85,B 0,C 180,E1 -9877.661,E2 -9877.661} C_VEL
LIN {X 0,Y 425.354,Z 368.497,A -85,B 0,C 180,E1 -9880.704,E2 -9880.704} C_VEL
LIN {X 0,Y 425.38,Z 368.495,A -85,B 0,C 180,E1 -9883.688,E2 -9883.688} C_VEL
LIN {X 0,Y 425.422,Z 368.491,A -85,B 0,C 180,E1 -9887.599,E2 -9887.599} C_VEL
LIN {X 0,Y 425.434,Z 368.491,A -85,B 0,C 180,E1 -9891.45,E2 -9891.45} C_VEL
LIN {X 0,Y 425.546,Z 368.469,A -85,B 0,C 180,E1 -9894.313,E2 -9894.313} C_VEL
LIN {X 0,Y 425.567,Z 368.469,A -85,B 0,C 180,E1 -9898.107,E2 -9898.107} C_VEL
LIN {X 0,Y 425.696,Z 368.454,A -85,B 0,C 180,E1 -9900,E2 -9900} C_VEL
LIN {X 0,Y 425.55,Z 368.474,A -85,B 0,C 180,E1 -9902.84,E2 -9902.84} C_VEL
LIN {X 0,Y 425.521,Z 368.482,A -85,B 0,C 180,E1 -9906.658,E2 -9906.658} C_VEL
LIN {X 0,Y 425.394,Z 368.492,A -85,B 0,C 180,E1 -9909.51,E2 -9909.51} C_VEL
LIN {X 0,Y 425.385,Z 368.495,A -85,B 0,C 180,E1 -9912.904,E2 -9912.904} C_VEL
LIN {X 0,Y 425.354,Z 368.499,A -85,B 0,C 180,E1 -9916.606,E2 -9916.606} C_VEL
LIN {X 0,Y 425.321,Z 368.502,A -85,B 0,C 180,E1 -9919.636,E2 -9919.636} C_VEL
LIN {X 0,Y 425.3,Z 368.505,A -85,B 0,C 180,E1 -9923.366,E2 -9923.366} C_VEL
LIN {X 0,Y 425.343,Z 368.491,A -85,B 0,C 180,E1 -9926.845,E2 -9926.845} C_VEL
LIN {X 0,Y 425.285,Z 368.508,A -85,B 0,C 180,E1 -9929.72,E2 -9929.72} C_VEL
LIN {X 0,Y 425.277,Z 368.508,A -85,B 0,C 180,E1 -9933.049,E2 -9933.049} C_VEL
LIN {X 0,Y 425.281,Z 368.513,A -85,B 0,C 180,E1 -9935.93,E2 -9935.93} C_VEL
LIN {X 0,Y 425.307,Z 368.504,A -85,B 0,C 180,E1 -9939.047,E2 -9939.047} C_VEL
LIN {X 0,Y 425.329,Z 368.501,A -85,B 0,C 180,E1 -9942.647,E2 -9942.647} C_VEL
LIN {X 0,Y 425.293,Z 368.511,A -85,B 0,C 180,E1 -9945.283,E2 -9945.283} C_VEL
LIN {X 0,Y 425.303,Z 368.509,A -85,B 0,C 180,E1 -9948.626,E2 -9948.626} C_VEL
LIN {X 0,Y 425.324,Z 368.505,A -85,B 0,C 180,E1 -9951.105,E2 -9951.105} C_VEL
LIN {X 0,Y 425.301,Z 368.508,A -85,B 0,C 180,E1 -9954.665,E2 -9954.665} C_VEL
LIN {X 0,Y 425.277,Z 368.512,A -85,B 0,C 180,E1 -9958.075,E2 -9958.075} C_VEL
LIN {X 0,Y 425.32,Z 368.517,A -85,B 0,C 180,E1 -9958.912,E2 -9958.912} C_VEL
LIN {X 0,Y 426.949,Z 376.865,A -85,B 0,C 180,E1 -9961.144,E2 -9961.144} C_VEL
LIN {X 0,Y 427.277,Z 380.617,A -85,B 0,C 180,E1 -9962.067,E2 -9962.067} C_VEL
LIN {X 0,Y 431.494,Z 398.452,A -85,B 0,C 180,E1 -9962.602,E2 -9962.602} C_VEL
LIN {X 0,Y 430.323,Z 487.047,A -85,B 0,C 180,E1 -9964.116,E2 -9964.116} C_VEL
LIN {X 0,Y 429.95,Z 499.386,A -85,B 0,C 180,E1 -9964.499,E2 -9964.499} C_VEL
LIN {X 0,Y 429.469,Z 511.952,A -85,B 0,C 180,E1 -9965.079,E2 -9965.079} C_VEL
LIN {X 0,Y 428.861,Z 523.741,A -85,B 0,C 180,E1 -9965.815,E2 -9965.815} C_VEL
LIN {X 0,Y 428.151,Z 535.713,A -85,B 0,C 180,E1 -9966.8,E2 -9966.8} C_VEL
LIN {X 0,Y 427.346,Z 546.382,A -85,B 0,C 180,E1 -9967.902,E2 -9967.902} C_VEL
LIN {X 0,Y 426.709,Z 555.046,A -85,B 0,C 180,E1 -9969.009,E2 -9969.009} C_VEL
LIN {X 0,Y 425.978,Z 563.842,A -85,B 0,C 180,E1 -9970.393,E2 -9970.393} C_VEL
LIN {X 0,Y 425.367,Z 571.768,A -85,B 0,C 180,E1 -9971.954,E2 -9971.954} C_VEL
LIN {X 0,Y 424.995,Z 576.939,A -85,B 0,C 180,E1 -9973.228,E2 -9973.228} C_VEL
LIN {X 0,Y 424.673,Z 581.56,A -85,B 0,C 180,E1 -9974.646,E2 -9974.646} C_VEL
LIN {X 0,Y 424.42,Z 585.205,A -85,B 0,C 180,E1 -9976.107,E2 -9976.107} C_VEL
LIN {X 0,Y 424.264,Z 588.124,A -85,B 0,C 180,E1 -9977.783,E2 -9977.783} C_VEL
LIN {X 0,Y 424.131,Z 589.767,A -85,B 0,C 180,E1 -9979.498,E2 -9979.498} C_VEL
LIN {X 0,Y 424.112,Z 589.839,A -85,B 0,C 180,E1 -9979.694,E2 -9979.694} C_VEL
LIN {X 0,Y 423.418,Z 590.176,A -85,B 0,C 180,E1 -9980.486,E2 -9980.486} C_VEL
LIN {X 0,Y 420.606,Z 590.144,A -85,B 0,C 180,E1 -9981.777,E2 -9981.777} C_VEL
LIN {X 0,Y 418.259,Z 589.614,A -85,B 0,C 180,E1 -9982.816,E2 -9982.816} C_VEL
LIN {X 0,Y 417.258,Z 588.835,A -85,B 0,C 180,E1 -9983.611,E2 -9983.611} C_VEL
LIN {X 0,Y 417.179,Z 588.496,A -85,B 0,C 180,E1 -9983.879,E2 -9983.879} C_VEL
LIN {X 0,Y 417.215,Z 585.509,A -85,B 0,C 180,E1 -9985.653,E2 -9985.653} C_VEL
LIN {X 0,Y 417.472,Z 581.936,A -85,B 0,C 180,E1 -9987.105,E2 -9987.105} C_VEL
LIN {X 0,Y 417.628,Z 577.286,A -85,B 0,C 180,E1 -9988.554,E2 -9988.554} C_VEL
LIN {X 0,Y 418.168,Z 570.275,A -85,B 0,C 180,E1 -9990.241,E2 -9990.241} C_VEL
LIN {X 0,Y 418.66,Z 562.695,A -85,B 0,C 180,E1 -9991.683,E2 -9991.683} C_VEL
LIN {X 0,Y 419.333,Z 553.173,A -85,B 0,C 180,E1 -9993.122,E2 -9993.122} C_VEL
LIN {X 0,Y 419.923,Z 543.379,A -85,B 0,C 180,E1 -9994.319,E2 -9994.319} C_VEL
LIN {X 0,Y 420.66,Z 532.332,A -85,B 0,C 180,E1 -9995.392,E2 -9995.392} C_VEL
LIN {X 0,Y 421.286,Z 521.531,A -85,B 0,C 180,E1 -9996.225,E2 -9996.225} C_VEL
LIN {X 0,Y 421.722,Z 509.66,A -85,B 0,C 180,E1 -9996.939,E2 -9996.939} C_VEL
LIN {X 0,Y 422.152,Z 496.626,A -85,B 0,C 180,E1 -9997.503,E2 -9997.503} C_VEL
LIN {X 0,Y 422.435,Z 483.594,A -85,B 0,C 180,E1 -9997.859,E2 -9997.859} C_VEL
LIN {X 0,Y 423.472,Z 398.571,A -85,B 0,C 180,E1 -9999.301,E2 -9999.301} C_VEL
LIN {X 0,Y 419.809,Z 380.459,A -85,B 0,C 180,E1 -9999.774,E2 -9999.774} C_VEL
LIN {X 0,Y 419.384,Z 375.092,A -85,B 0,C 180,E1 -10001.111,E2 -10001.111} C_VEL
LIN {X 0,Y 418.378,Z 369.373,A -85,B 0,C 180,E1 -10002.613,E2 -10002.613} C_VEL
LIN {X 0,Y 418.316,Z 369.377,A -85,B 0,C 180,E1 -10005.593,E2 -10005.593} C_VEL
LIN {X 0,Y 418.288,Z 369.382,A -85,B 0,C 180,E1 -10008.616,E2 -10008.616} C_VEL
LIN {X 0,Y 418.238,Z 369.385,A -85,B 0,C 180,E1 -10011.696,E2 -10011.696} C_VEL
LIN {X 0,Y 418.287,Z 369.38,A -85,B 0,C 180,E1 -10014.864,E2 -10014.864} C_VEL
LIN {X 0,Y 418.298,Z 369.38,A -85,B 0,C 180,E1 -10018.062,E2 -10018.062} C_VEL
LIN {X 0,Y 418.218,Z 369.387,A -85,B 0,C 180,E1 -10021.395,E2 -10021.395} C_VEL
LIN {X 0,Y 418.267,Z 369.384,A -85,B 0,C 180,E1 -10024.579,E2 -10024.579} C_VEL
LIN {X 0,Y 418.235,Z 369.387,A -85,B 0,C 180,E1 -10027.834,E2 -10027.834} C_VEL
LIN {X 0,Y 418.221,Z 369.389,A -85,B 0,C 180,E1 -10030.947,E2 -10030.947} C_VEL
LIN {X 0,Y 418.208,Z 369.39,A -85,B 0,C 180,E1 -10033.728,E2 -10033.728} C_VEL
LIN {X 0,Y 418.281,Z 369.382,A -85,B 0,C 180,E1 -10036.457,E2 -10036.457} C_VEL
LIN {X 0,Y 418.264,Z 369.382,A -85,B 0,C 180,E1 -10039.122,E2 -10039.122} C_VEL
LIN {X 0,Y 418.234,Z 369.39,A -85,B 0,C 180,E1 -10042.164,E2 -10042.164} C_VEL
LIN {X 0,Y 418.261,Z 369.383,A -85,B 0,C 180,E1 -10045.419,E2 -10045.419} C_VEL
LIN {X 0,Y 418.207,Z 369.391,A -85,B 0,C 180,E1 -10048.603,E2 -10048.603} C_VEL
LIN {X 0,Y 418.286,Z 369.384,A -85,B 0,C 180,E1 -10051.936,E2 -10051.936} C_VEL
LIN {X 0,Y 418.284,Z 369.38,A -85,B 0,C 180,E1 -10055.162,E2 -10055.162} C_VEL
LIN {X 0,Y 418.249,Z 369.387,A -85,B 0,C 180,E1 -10058.304,E2 -10058.304} C_VEL
LIN {X 0,Y 418.277,Z 369.381,A -85,B 0,C 180,E1 -10061.382,E2 -10061.382} C_VEL
LIN {X 0,Y 418.296,Z 369.381,A -85,B 0,C 180,E1 -10064.405,E2 -10064.405} C_VEL
LIN {X 0,Y 418.364,Z 369.371,A -85,B 0,C 180,E1 -10067.386,E2 -10067.386} C_VEL
LIN {X 0,Y 418.353,Z 369.374,A -85,B 0,C 180,E1 -10070.329,E2 -10070.329} C_VEL
LIN {X 0,Y 418.485,Z 369.355,A -85,B 0,C 180,E1 -10073.249,E2 -10073.249} C_VEL
LIN {X 0,Y 418.335,Z 369.374,A -85,B 0,C 180,E1 -10075.181,E2 -10075.181} C_VEL
LIN {X 0,Y 418.537,Z 369.351,A -85,B 0,C 180,E1 -10078.075,E2 -10078.075} C_VEL
LIN {X 0,Y 418.666,Z 369.335,A -85,B 0,C 180,E1 -10080,E2 -10080} C_VEL
LIN {X 0,Y 418.504,Z 369.353,A -85,B 0,C 180,E1 -10082.888,E2 -10082.888} C_VEL
LIN {X 0,Y 418.486,Z 369.356,A -85,B 0,C 180,E1 -10086.751,E2 -10086.751} C_VEL
LIN {X 0,Y 418.352,Z 369.374,A -85,B 0,C 180,E1 -10089.671,E2 -10089.671} C_VEL
LIN {X 0,Y 418.347,Z 369.372,A -85,B 0,C 180,E1 -10093.007,E2 -10093.007} C_VEL
LIN {X 0,Y 418.304,Z 369.378,A -85,B 0,C 180,E1 -10096.736,E2 -10096.736} C_VEL
LIN {X 0,Y 418.294,Z 369.381,A -85,B 0,C 180,E1 -10099.803,E2 -10099.803} C_VEL
LIN {X 0,Y 418.235,Z 369.386,A -85,B 0,C 180,E1 -10102.736,E2 -10102.736} C_VEL
LIN {X 0,Y 418.264,Z 369.385,A -85,B 0,C 180,E1 -10105.904,E2 -10105.904} C_VEL
LIN {X 0,Y 418.258,Z 369.383,A -85,B 0,C 180,E1 -10109.162,E2 -10109.162} C_VEL
LIN {X 0,Y 418.251,Z 369.384,A -85,B 0,C 180,E1 -10112.845,E2 -10112.845} C_VEL
LIN {X 0,Y 418.243,Z 369.388,A -85,B 0,C 180,E1 -10116.239,E2 -10116.239} C_VEL
LIN {X 0,Y 418.261,Z 369.385,A -85,B 0,C 180,E1 -10119.681,E2 -10119.681} C_VEL
LIN {X 0,Y 418.28,Z 369.382,A -85,B 0,C 180,E1 -10122.33,E2 -10122.33} C_VEL
LIN {X 0,Y 418.247,Z 369.384,A -85,B 0,C 180,E1 -10125.112,E2 -10125.112} C_VEL
LIN {X 0,Y 418.236,Z 369.389,A -85,B 0,C 180,E1 -10127.768,E2 -10127.768} C_VEL
LIN {X 0,Y 418.254,Z 369.385,A -85,B 0,C 180,E1 -10131.559,E2 -10131.559} C_VEL
LIN {X 0,Y 418.258,Z 369.382,A -85,B 0,C 180,E1 -10135.16,E2 -10135.16} C_VEL
LIN {X 0,Y 418.248,Z 369.385,A -85,B 0,C 180,E1 -10137.473,E2 -10137.473} C_VEL
LIN {X 0,Y 418.276,Z 369.383,A -85,B 0,C 180,E1 -10140.894,E2 -10140.894} C_VEL
LIN {X 0,Y 418.347,Z 369.591,A -85,B 0,C 180,E1 -10142.065,E2 -10142.065} C_VEL
LIN {X 0,Y 421.017,Z 382.993,A -85,B 0,C 180,E1 -10144.848,E2 -10144.848} C_VEL
LIN {X 0,Y 421.194,Z 386.867,A -85,B 0,C 180,E1 -10145.609,E2 -10145.609} C_VEL
LIN {X 0,Y 420.086,Z 404.354,A -85,B 0,C 180,E1 -10148.919,E2 -10148.919} C_VEL
LIN {X 0,Y 419.39,Z 416.575,A -85,B 0,C 180,E1 -10151.213,E2 -10151.213} C_VEL
LIN {X 0,Y 423.169,Z 444.306,A -85,B 0,C 180,E1 -10151.848,E2 -10151.848} C_VEL
LIN {X 0,Y 422.301,Z 525.892,A -85,B 0,C 180,E1 -10153.255,E2 -10153.255} C_VEL
LIN {X 0,Y 421.75,Z 539.74,A -85,B 0,C 180,E1 -10153.699,E2 -10153.699} C_VEL
LIN {X 0,Y 421.157,Z 552.678,A -85,B 0,C 180,E1 -10154.329,E2 -10154.329} C_VEL
LIN {X 0,Y 420.389,Z 564.472,A -85,B 0,C 180,E1 -10155.106,E2 -10155.106} C_VEL
LIN {X 0,Y 419.708,Z 575.87,A -85,B 0,C 180,E1 -10156.072,E2 -10156.072} C_VEL
LIN {X 0,Y 419.088,Z 586.125,A -85,B 0,C 180,E1 -10157.162,E2 -10157.162} C_VEL
LIN {X 0,Y 418.488,Z 595.35,A -85,B 0,C 180,E1 -10158.374,E2 -10158.374} C_VEL
LIN {X 0,Y 417.87,Z 604.331,A -85,B 0,C 180,E1 -10159.829,E2 -10159.829} C_VEL
LIN {X 0,Y 417.514,Z 611.551,A -85,B 0,C 180,E1 -10161.287,E2 -10161.287} C_VEL
LIN {X 0,Y 417.265,Z 617.299,A -85,B 0,C 180,E1 -10162.743,E2 -10162.743} C_VEL
LIN {X 0,Y 417.102,Z 621.82,A -85,B 0,C 180,E1 -10164.198,E2 -10164.198} C_VEL
LIN {X 0,Y 417.14,Z 624.208,A -85,B 0,C 180,E1 -10165.168,E2 -10165.168} C_VEL
LIN {X 0,Y 417.037,Z 626.152,A -85,B 0,C 180,E1 -10166.135,E2 -10166.135} C_VEL
LIN {X 0,Y 417.108,Z 627.678,A -85,B 0,C 180,E1 -10167.103,E2 -10167.103} C_VEL
LIN {X 0,Y 417.093,Z 628.742,A -85,B 0,C 180,E1 -10168.069,E2 -10168.069} C_VEL
LIN {X 0,Y 417.052,Z 629.687,A -85,B 0,C 180,E1 -10170,E2 -10170} C_VEL
LIN {X 0,Y 417.055,Z 629.573,A -85,B 0,C 180,E1 -10170.966,E2 -10170.966} C_VEL
LIN {X 0,Y 417.091,Z 629.026,A -85,B 0,C 180,E1 -10171.931,E2 -10171.931} C_VEL
LIN {X 0,Y 417.072,Z 628.08,A -85,B 0,C 180,E1 -10172.898,E2 -10172.898} C_VEL
LIN {X 0,Y 417.113,Z 624.988,A -85,B 0,C 180,E1 -10174.833,E2 -10174.833} C_VEL
LIN {X 0,Y 417.142,Z 621.556,A -85,B 0,C 180,E1 -10176.262,E2 -10176.262} C_VEL
LIN {X 0,Y 417.349,Z 616.913,A -85,B 0,C 180,E1 -10177.742,E2 -10177.742} C_VEL
LIN {X 0,Y 417.731,Z 610,A -85,B 0,C 180,E1 -10179.441,E2 -10179.441} C_VEL
LIN {X 0,Y 418.253,Z 602.531,A -85,B 0,C 180,E1 -10180.896,E2 -10180.896} C_VEL
LIN {X 0,Y 418.906,Z 594.935,A -85,B 0,C 180,E1 -10182.105,E2 -10182.105} C_VEL
LIN {X 0,Y 419.57,Z 585.755,A -85,B 0,C 180,E1 -10183.316,E2 -10183.316} C_VEL
LIN {X 0,Y 420.328,Z 575.478,A -85,B 0,C 180,E1 -10184.41,E2 -10184.41} C_VEL
LIN {X 0,Y 421.164,Z 564.313,A -85,B 0,C 180,E1 -10185.361,E2 -10185.361} C_VEL
LIN {X 0,Y 421.98,Z 552.658,A -85,B 0,C 180,E1 -10186.136,E2 -10186.136} C_VEL
LIN {X 0,Y 422.698,Z 540.772,A -85,B 0,C 180,E1 -10186.729,E2 -10186.729} C_VEL
LIN {X 0,Y 423.295,Z 527.751,A -85,B 0,C 180,E1 -10187.171,E2 -10187.171} C_VEL
LIN {X 0,Y 423.585,Z 508.298,A -85,B 0,C 180,E1 -10187.552,E2 -10187.552} C_VEL
LIN {X 0,Y 424.252,Z 443.024,A -85,B 0,C 180,E1 -10188.677,E2 -10188.677} C_VEL
LIN {X 0,Y 420.597,Z 420.093,A -85,B 0,C 180,E1 -10189.277,E2 -10189.277} C_VEL
LIN {X 0,Y 419.922,Z 416.211,A -85,B 0,C 180,E1 -10189.401,E2 -10189.401} C_VEL
LIN {X 0,Y 421.128,Z 398.596,A -85,B 0,C 180,E1 -10192.797,E2 -10192.797} C_VEL
LIN {X 0,Y 421.942,Z 387.987,A -85,B 0,C 180,E1 -10194.87,E2 -10194.87} C_VEL
LIN {X 0,Y 420.988,Z 381.462,A -85,B 0,C 180,E1 -10196.255,E2 -10196.255} C_VEL
LIN {X 0,Y 418.66,Z 371.036,A -85,B 0,C 180,E1 -10198.582,E2 -10198.582} C_VEL
LIN {X 0,Y 418.295,Z 369.38,A -85,B 0,C 180,E1 -10199.015,E2 -10199.015} C_VEL
LIN {X 0,Y 418.248,Z 369.386,A -85,B 0,C 180,E1 -10202.527,E2 -10202.527} C_VEL
LIN {X 0,Y 418.258,Z 369.384,A -85,B 0,C 180,E1 -10204.84,E2 -10204.84} C_VEL
LIN {X 0,Y 418.258,Z 369.384,A -85,B 0,C 180,E1 -10208.44,E2 -10208.44} C_VEL
LIN {X 0,Y 418.22,Z 369.385,A -85,B 0,C 180,E1 -10210.947,E2 -10210.947} C_VEL
LIN {X 0,Y 418.206,Z 369.391,A -85,B 0,C 180,E1 -10213.729,E2 -10213.729} C_VEL
LIN {X 0,Y 418.268,Z 369.378,A -85,B 0,C 180,E1 -10216.456,E2 -10216.456} C_VEL
LIN {X 0,Y 418.262,Z 369.38,A -85,B 0,C 180,E1 -10219.123,E2 -10219.123} C_VEL
LIN {X 0,Y 418.232,Z 369.384,A -85,B 0,C 180,E1 -10222.164,E2 -10222.164} C_VEL
